// TIA Portal project "EdgeHowTos_V19" (V19)

(* hardware
DEVICE "S71500/ET200MP station_1"  S7-1500 station
   slot 0: "Rail_0"  Rack  6ES7 590-1***0-0AA0
   slot 1: "Tank application"  CPU 1513-1 PN  6ES7 513-1AL02-0AB0  V2.8
      slot 3: "CPU display_1"  6ES7591-1AA00-0AA0
      slot 32768: "PROFINET interface_1"  X1
         slot 32769: "Port_1"  X1 P1
         slot 32770: "Port_2"  X1 P2
      slot 34817: "Virtual CP interface port_1"  Virtual CP interface port  Virtual CP interface port
DEVICE "TP900"  TP900 Comfort
   slot 0: "TP900"  TP900 Comfort  6AV2 124-0JC01-0AX0  16.0.0.0
   slot 1: "HMI_RT_5"  TP900 Comfort  6AV2 124-0JC01-0AX0  16.0.0.0
   slot 5: "TP900._CP_1"  PROFINET Interface  16.0.0.0
      slot 1: "PROFINET Interface_1"  PROFINET Interface
         slot 1: "Port_1"  Port
         slot 2: "Port_2"  Port
   slot 7: "TP900.I/DP_CP_1"  MPI/DP Interface  16.0.0.0
DEVICE "MTP1500"  MTP1500 Unified Comfort
   slot 0: "0"  MTP1500 Unified Comfort  6AV2 128-3QB06-0AXx  19.0.0.0
   slot 1: "MTP1500_Runtime"  MTP1500 Unified Comfort  6AV2 128-3QB06-0AXx  19.0.0.0
   slot 5: "0.IE_CP_1"  PROFINET Interface  19.0.0.0
      slot 1: "PROFINET Interface_1"  PROFINET Interface
         slot 1: "Port_1"  Port
         slot 2: "Port_2"  Port
   slot 6: "0.IE_CP_2"  PROFINET Interface  19.0.0.0
      slot 1: "PROFINET Interface_GBit"  PROFINET Interface
         slot 1: "Port_1"  Port
*)

// ===== PLC "Tank application"  CPU 1513-1 PN =====

VAR_GLOBAL   // PLC tag table "Default tag table"
   "Manipulator" AT %MW0 : Int;
END_VAR

VAR_GLOBAL CONSTANT   // PLC tag table "Default tag table"
   "STATE_FILL_TANK" : Int := 1;
   "STATE_HEAT_TANK" : Int := 2;
   "STATE_FILL_BOTTLE" : Int := 3;
   "STATE_SHIFT_BOTTLE" : Int := 4;
   "STATE_STOP" : Int := 5;
   "STATE_RESET" : Int := 6;
   "STATE_ERROR" : Int := 7;
   "ERROR_0_NoError" : UInt := 8000;
   "ERROR_1_BottleInWrongPosition" : UInt := 8001;
   "ERROR_2_CrackedBottleDetected" : UInt := 8002;
   "ERROR_3_NoBottleOnTheConveyor" : UInt := 8003;
   "ERROR_4_WrongBottleDetected" : UInt := 8004;
   "ERROR_5_ConveyorMalfunction" : UInt := 8005;
   "ERROR_6_FillerMalfunction" : UInt := 8006;
   "ERROR_7_ValveBlocked" : UInt := 8007;
   "ERROR_8_NoFlowInMainPipe" : UInt := 8008;
   "ERROR_9_GenericError_CheckPlcBuffer" : UInt := 8009;
   "ERROR_10_GenericError_CheckAlarmBuffer" : UInt := 8010;
   "ERROR_11_GenericError_ContactWithSupplier" : UInt := 8011;
   "OEE_ERROR_1_BottleInWrongPosition" : UInt := 4;
   "OEE_ERROR_10_GenericError_CheckAlarmBuffer" : UInt := 13;
   "OEE_ERROR_11_GenericError_ContactWithSupplier" : UInt := 14;
   "OEE_ERROR_2_CrackedBottleDetected" : UInt := 5;
   "OEE_ERROR_3_NoBottleOnTheConveyor" : UInt := 6;
   "OEE_ERROR_4_WrongBottleDetected" : UInt := 7;
   "OEE_ERROR_5_ConveyorMalfunction" : UInt := 8;
   "OEE_ERROR_6_FillerMalfunction" : UInt := 9;
   "OEE_ERROR_7_ValveBlocked" : UInt := 10;
   "OEE_ERROR_8_NoFlowInMainPipe" : UInt := 11;
   "OEE_ERROR_9_GenericError_CheckPlcBuffer" : UInt := 12;
   "OEE_PRODUCTION" : UInt := 1;
   "OEE_PLANNED_DOWN" : UInt := 2;
   "OEE_UNPLANNED_DOWN" : UInt := 3;
END_VAR

TYPE "typeHmi"
   STRUCT
      HMI_Start : Bool;   // trigger from hmi to start
      HMI_Stop : Bool;   // trigger from hmi to stop
      HMI_Reset : Bool;   // trigger from hmi to reset
      HMI_NextBottle : Bool;   // trigger from hmi to shift bottle
      HMI_Error : Bool;   // trigger from hmi to generate error
      HMI_InstallFillingPump : Bool;   // trigger from hmi to install filling pump
      HMI_RenewHeatingElement : Bool;   // trigger from hmi to renew heating element
   END_STRUCT;
END_TYPE

TYPE "typeApp"
   STRUCT
      APP_Start : Bool;   // trigger from app to start
      APP_Stop : Bool;   // trigger from app to stop
      APP_Reset : Bool;   // trigger from app to reset
      APP_QRCode : String;   // string from app containing QR code (scanning app)
      APP_ErrorSimulation : Bool;   // activate automatically error simulation (true = active)
      APP_Error : Bool;   // generate a manual error (true = error)
      APP_Alarm : Bool;   // trigger from app to generate program alarm
   END_STRUCT;
END_TYPE

TYPE "typeSignals"
   STRUCT
      tankSignals : Struct
         actLevel : Real;   // actual level of tank [l]
         maxLevel : Bool;   // max level of tank reached
         actPressure : Real;   // actual pressure of tank [hPa]
         actTemperature : Real;   // actual temperature of tank [°C]
         maxTemperature : Bool;   // max level of temperature reached
      END_STRUCT;
      bottleSignals : Struct
         actLevel : Real;   // actual level of current bottle [l]
         maxLevel : Bool;   // max level of bottle reached
         outputTank : Real;   // Vout of Tank / Vin of bottle [m³/s]
      END_STRUCT;
      energySignals : Struct
         energyConsumptionFillingTank : Real;   // energy consumption during filling tank [Wh]
         waterConsumptionFillingTank : Real;   // water consumption during filling tank [l]
         energyConsumptionHeatingTank : Real;   // energy consumption during heating tank [Wh]
         energyConsumptionFillingBottles : Real;   // energy consumption during filling bottles [Wh]
         gasConsumptionHeatingTank : Real;   // gas consumption during heating tank [Wh]
      END_STRUCT;
      energySignalsPerState : Struct
         stateId : UInt;   // ID per standart state
         energyConsumptionStatePoweringUp : Real;   // energy consumption during state powering up [kWh]
         energyConsumptionStatePoweringDown : Real;   // energy consumption during state powering down [kWh]
         energyConsumptionStateOff : Real;   // energy consumption during state off [kWh]
         energyConsumptionStateStandby : Real;   // energy consumption during state standby [kWh]
         energyConsumptionStateOperational : Real;   // energy consumption during state operational [kWh]
         energyConsumptionStateWorking : Real;   // energy consumption during state working [kWh]
         energyConsumptionStatesTotal : Real;   // total energy consumption of states [kWh]
      END_STRUCT;
      alarm : Word;   // alarm bit
      errorCode : UInt;   // error code
   END_STRUCT;
END_TYPE

TYPE "typeOperate"
   STRUCT
      extModeActive : Bool := false;   // true = activate external model / simulation
      state : "typeState";   // operating state
      machineState : Int := 0;   // machine production state (1 = filling tank, 2 = heating tank, 3 = filling bottle, 4 = shifting bottle, 5 = stop, 6 = reset)
      machineStateOEE : Int := 0;   // machine OEE state (1 = production, 2 = planned downtime, 3 = unplanned downtime)
   END_STRUCT;
END_TYPE

TYPE "typeModel"
   STRUCT
      cycleTime : Real;   // cycle time[s]
      tank : Struct   // model struct of tank
         AT : Real;   // surface area of tank [m²]
         H : Real;   // high of tank [m]
         Vin : Real;   // incoming volume flow [l/min]
         maxLevel : Real;   // max level of tank [m³]
         roomTemperature : Real;   // room temperature of tank [°C]
         maxTemperature : Real;   // max temperature of tank [°C]
         density : Real;   // liquid density [kg/m³]
      END_STRUCT;
      bottle : Struct   // model struct of bottle
         maxLevel : Real;   // max level of bottle [m³]
         AB : Real;   // surface area of filling hole to fill bottle [m²]
         shiftingCycle : UInt;   // bottle shifting cycle
      END_STRUCT;
   END_STRUCT;
END_TYPE

TYPE "typeProcess"
   STRUCT
      productId : String;   // product id of current bottle
      numberProduced : UDInt;   // number of filled bottles
      numberFaulty : UDInt;   // number of faulty bottles
      numberGood : UDInt;   // number of good bottles
      batchId : UDInt;   // batch id (according to tank filling)
      productTypeId : UInt;   // type id - for generating of the serial number and QR code
      productTypeName : String;   // type name of product
      productSerialNumber : String;   // serial number per product
      productQRCode : USInt;   // qr code per product
      speedActual : UDInt;   // actual production speed (pcs/h)
      speedTarget : UDInt;   // target production speed (pcs/h)
   END_STRUCT;
END_TYPE

TYPE "typeState"
   STRUCT
      FillingTank : Bool;   // filling tank
      HeatingTank : Bool;   // heating tank
      FillingBottle : Bool;   // filling bottle
      ShiftingBottle : Bool;   // shifting bottle
      Stop : Bool;   // stop filling application
      Reset : Bool;   // reset application
      Error : Bool;   // error within filling application
   END_STRUCT;
END_TYPE

TYPE "typeInfo"
   STRUCT
      "version" : String;   // current version of the project
      "date" : String;   // last change date of the project
   END_STRUCT;
END_TYPE

TYPE "typeError"
   STRUCT
      errorTrigger : Bool := false;   // manually trigger error simulation
      errorDuration : Time := T#300s;   // error duration for simulation
   END_STRUCT;
END_TYPE

TYPE "typeCIP"
   STRUCT
      cipStartTime : Time_Of_Day := TOD#22:00:00;   // CIP start time 1x per day
      cipActive : Bool;   // Activate/deactivate the CIP process
      cipId : Int;   // CIP id
      cipProcess : String;   // CIP process (full wash, quick wash)
      cipStep : String;   // CIP step
      cipTemperature : Real;   // CIP temperature
      cipConcentration : Real;   // CIP concentration
      cipFlowrate : Real;   // CIP flowrate
      cipStep1 : Bool;   // Step 1 active
      cipStep2 : Bool;   // Step 2 active
      cipStep3 : Bool;   // Step 3 active
      cipStep4 : Bool;   // Step 4 active
   END_STRUCT;
END_TYPE

DATA_BLOCK "GDB"   // DB1
{ S7_Optimized_Access := 'FALSE' }
VERSION : 0.1
   VAR
      operate : "typeOperate";   // application operation
      model : "typeModel";   // model parameter
      externalSignals : "typeSignals";   // signals from external model
      signals : "typeSignals";   // current signals from tank and bottle
      process : "typeProcess";   // current process information
      hmiSignals : "typeHmi";   // signals from hmi
      appSignals : "typeApp";   // signals from edge app
      projectInfo : "typeInfo";   // infos regarding this TIA project
      errors : "typeError";   // parameter for error simulation
      cip : "typeCIP";   // parameter for cip simulation (tank cleaning)
   END_VAR
BEGIN
   model.tank.H := 2.0;
   model.tank.AT := 0.8;
   operate.extModeActive := false;
   model.tank.maxTemperature := 80.0;
   model.tank.maxLevel := 1.6;
   model.bottle.maxLevel := 0.001;
   model.cycleTime := 0.005;
   model.tank.roomTemperature := 20.0;
   model.tank.Vin := 500.0;
   model.bottle.AB := 5.0E-06;
   process.productId := '';
   process.numberProduced := 0;
   process.numberFaulty := 0;
   model.tank.density := 997.0;
   hmiSignals.HMI_Start := true;
   projectInfo."version" := 'V4.0';
   projectInfo."date" := '2025-07-01';
   errors.errorDuration := T#10m;
   model.bottle.shiftingCycle := 50;
   appSignals.APP_ErrorSimulation := true;
   process.speedActual := 3700;
   process.speedTarget := 4000;
END_DATA_BLOCK

DATA_BLOCK "DB_1_Sequence"   // DB2
{ S7_Optimized_Access := 'TRUE' }
VERSION : 0.1
// stored: InstanceOfName FB_1_Sequence
"FB_1_Sequence"
BEGIN
END_DATA_BLOCK

DATA_BLOCK "DB_2_Filling_DB"   // DB3
{ S7_Optimized_Access := 'TRUE' }
VERSION : 0.1
// stored: InstanceOfName FB_2_Filling
"FB_2_Filling"
BEGIN
END_DATA_BLOCK

DATA_BLOCK "DB_3_Simulation"   // DB4
{ S7_Optimized_Access := 'TRUE' }
VERSION : 0.1
// stored: InstanceOfName FB_3_Simulation
"FB_3_Simulation"
BEGIN
END_DATA_BLOCK

DATA_BLOCK "Generate_Serial_Number_DB"   // DB6
{ S7_Optimized_Access := 'TRUE' }
VERSION : 0.1
// stored: InstanceOfName FB_Generate_Serial_Number
"FB_Generate_Serial_Number"
BEGIN
END_DATA_BLOCK

DATA_BLOCK "Block_1_DB"   // DB7
{ S7_Optimized_Access := 'TRUE' }
VERSION : 0.1
// stored: InstanceOfName FB_Prodiag
"FB_Prodiag"
BEGIN
END_DATA_BLOCK

DATA_BLOCK "DB_4_CIP_Simulation"   // DB11
{ S7_Optimized_Access := 'TRUE' }
VERSION : 0.1
// stored: InstanceOfName FB_4_CIP_Simulation
"FB_4_CIP_Simulation"
BEGIN
END_DATA_BLOCK

DATA_BLOCK "DB_5_CIP_Simulation_Graph"   // DB14
{ S7_Optimized_Access := 'TRUE' }
VERSION : 0.1
// stored: InstanceOfName FB_5_CIP_Simulation_Graph
"FB_5_CIP_Simulation_Graph"
BEGIN
END_DATA_BLOCK

// folder: System blocks/Program resources

DATA_BLOCK "IEC_Timer_CIP_Step2"   // DB12
{ S7_Optimized_Access := 'TRUE' }
AUTHOR : Simatic
FAMILY : IEC
NAME : IEC_TMR
VERSION : 1.0
// stored: InstanceOfName IEC_TIMER
"IEC_TIMER"
BEGIN
END_DATA_BLOCK

DATA_BLOCK "IEC_Timer_CIP_Init"   // DB15
{ S7_Optimized_Access := 'TRUE' }
AUTHOR : Simatic
FAMILY : IEC
NAME : IEC_TMR
VERSION : 1.0
// stored: InstanceOfName IEC_TIMER
"IEC_TIMER"
BEGIN
END_DATA_BLOCK

DATA_BLOCK "IEC_Timer_CIP_Step3"   // DB20
{ S7_Optimized_Access := 'TRUE' }
AUTHOR : Simatic
FAMILY : IEC
NAME : IEC_TMR
VERSION : 1.0
// stored: InstanceOfName IEC_TIMER
"IEC_TIMER"
BEGIN
END_DATA_BLOCK

DATA_BLOCK "IEC_Timer_CIP_Step4"   // DB21
{ S7_Optimized_Access := 'TRUE' }
AUTHOR : Simatic
FAMILY : IEC
NAME : IEC_TMR
VERSION : 1.0
// stored: InstanceOfName IEC_TIMER
"IEC_TIMER"
BEGIN
END_DATA_BLOCK

DATA_BLOCK "IEC_Timer_CIP_End"   // DB22
{ S7_Optimized_Access := 'TRUE' }
AUTHOR : Simatic
FAMILY : IEC
NAME : IEC_TMR
VERSION : 1.0
// stored: InstanceOfName IEC_TIMER
"IEC_TIMER"
BEGIN
END_DATA_BLOCK

// folder: (top level)

FUNCTION_BLOCK "FB_Generate_Serial_Number"   // FB1, LAD
{ S7_Optimized_Access := 'TRUE' }
VERSION : 0.1
   VAR_INPUT
      batchId : UDInt;
      productId : UDInt;
      productType : Int;
      trigger : Bool;
   END_VAR
   VAR_OUTPUT
      serialNumber : String;
      qrCode : USInt;
   END_VAR
   VAR
      sizeBatch : USInt;
      sizeId : USInt;
      retVal : USInt;
      dateString : String;
      batchString : String;
      productString : String;
      typeString : String;
      pTrigAux_1 : Bool;
   END_VAR
   VAR_TEMP
      localTime : DTL;
      qrNoTemp : String;
   END_VAR
   VAR_TEMP   // added for the SCL form of the ladder/FBD networks
      _w1 : Bool;
   END_VAR
BEGIN

REGION Network 1 (SCL)
   // get string size of batch ID
   "FC_2_GetStringSizeOfNumber"(number:=#batchId,
                                stringSize=>#sizeBatch);

   // get string size of prodcut ID
   "FC_2_GetStringSizeOfNumber"(number:=#productId,
                                stringSize=>#sizeId);
END_REGION

REGION Network 2
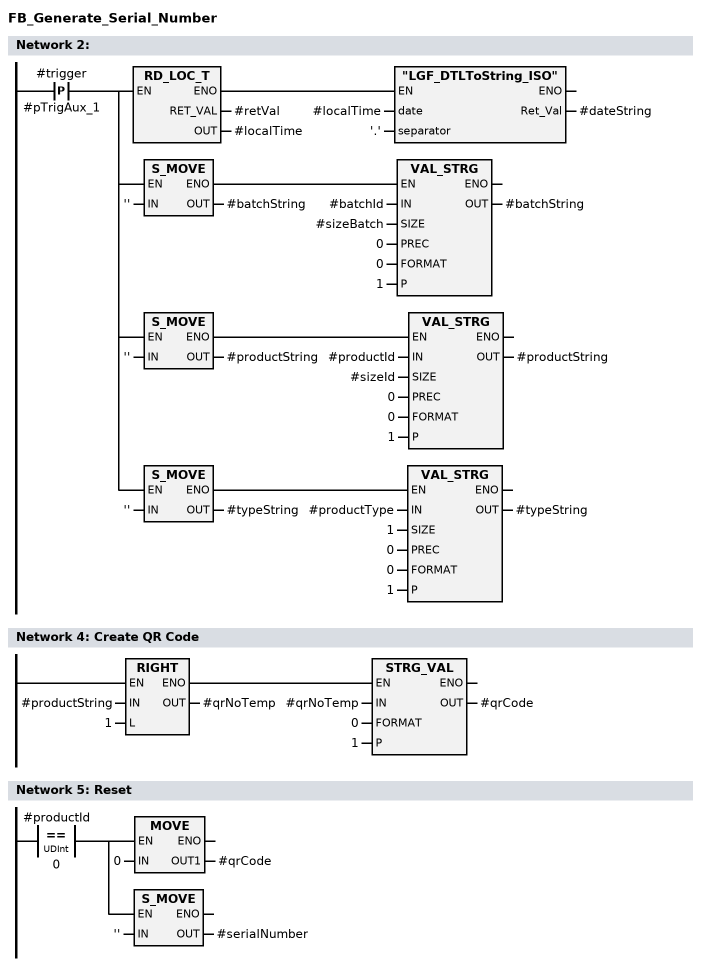
   // ENO of a box is taken as its EN; it also drops when the box reports an error
   #_w1 := #trigger AND NOT #pTrigAux_1;   // rising edge of #trigger
   #pTrigAux_1 := #trigger;
   IF #_w1 THEN
       #retVal := RD_LOC_T(OUT => #localTime);
       #dateString := "LGF_DTLToString_ISO"("date" := #localTime, separator := '.');
       #batchString := '';
       VAL_STRG(IN := #batchId, SIZE := #sizeBatch, PREC := 0, FORMAT := 0, P := 1, OUT => #batchString);
       #productString := '';
       VAL_STRG(IN := #productId, SIZE := #sizeId, PREC := 0, FORMAT := 0, P := 1, OUT => #productString);
       #typeString := '';
       VAL_STRG(IN := #productType, SIZE := 1, PREC := 0, FORMAT := 0, P := 1, OUT => #typeString);
   END_IF;
END_REGION

REGION Network 3 (SCL): Create serial number
   #serialNumber := CONCAT(
                            IN1 := REPLACE(IN1:=DELETE(IN:=#dateString, L:=13, P:=17), IN2:='/', L:=1, P:=11),
                            IN2 := '/',
                            IN3 := #typeString,
                            IN4 := '/',
                            IN5 := #batchString,
                            IN6 := '/',
                            IN7 := #productString
   );
END_REGION

REGION Network 4: Create QR Code
   #qrNoTemp := RIGHT(IN := #productString, L := 1);
   STRG_VAL(IN := #qrNoTemp, FORMAT := 0, P := 1, OUT => #qrCode);
END_REGION

REGION Network 5: Reset
   RUNG wire#powerrail
      { S7_Templates := "SrcType := UDInt" } EQ_Contact(in1 := #productId, in2 := 0)
      wire#w1
      Move(in := 0, out1 => #qrCode)
   END_RUNG
   RUNG wire#w1
      S_Move(in := '', out => #serialNumber)
   END_RUNG
   // the same network as SCL:
   IF #productId = 0 THEN
       #qrCode := 0;
       #serialNumber := '';
   END_IF;
END_REGION
END_FUNCTION_BLOCK

FUNCTION_BLOCK "FB_1_Sequence"   // FB2, FBD
{ S7_Optimized_Access := 'TRUE' }
VERSION : 0.1
   VAR_INPUT
      externalSignals : "typeSignals";   // signals from external model
   END_VAR
   VAR_IN_OUT
      model : "typeModel";   // model parameter
      operate : "typeOperate";   // application operation
      signals : "typeSignals";   // current signals from tank
      process : "typeProcess";   // current process information
      hmi : "typeHmi";   // signals from hmi
      app : "typeApp";   // signals from app
      errors : "typeError";
   END_VAR
   VAR
      statStart : Bool;   // trigger for start command
      statStop : Bool;   // trigger for stop command
      statReset : Bool;   // trigger for reset command
      statInit : Bool := true;   // helper variable to initialize some parameters
      statNextBottle : Bool;   // trigger to shift next bottle
      statError : Bool;   // trigger to set error
      statState : Int;   // memory for reactivating state after STOP
      statAlarm : Bool;   // trigger to generate program alarm
      statMemoryStart : Bool;
      statMemoryStop : Bool;
      statMemoryReset : Bool;
      statMemoryNextBottle : Bool;
      statMemoryError : Bool;
      statHmiStateStart : Bool;   // helper for hmi (true, if state 1-4)
      statShiftingTimer : Int;
      statShiftingTimerTrigger : Bool;
      statShiftingTrigger : Bool;
      statShiftingTimerDone : Bool;
      statHmiQrCodeReceived : Bool;
      statHMIQrCodeReceivedTrigger : Bool;
      statQrCodeTrigger : Bool;
      statTankEmpty : Bool;   // trigger when tank is empty
      statTankEmptyMemory : Bool;   // tank empty memory
      statOverflow : Bool;   // overflow of counter "numberProduced"
      statOverflowStartTrigger : Bool;   // trigger to start after overflow
      statOverflowStartMemory : Bool;
      Program_Alarm : Program_Alarm;
      statAssocValues : AssocValues;   // values for Gen_UsrMsg block
      statTriggerAlarm : Bool;
      statTriggerAlarmMemory : Bool;
      statErrorCodeOld : UInt;
   END_VAR
   VAR_TEMP
      tempQrCodeLen : Int;
      tempProgramAlarmError : Bool;
      tempProgramAlarmStatus : Word;
      tempAlarmStateError : Bool;
      tempAlarmStateStatus : Word;
      tempProgramAlarmError2 : Bool;
      tempProgramAlarmStatus2 : Word;
      tempAlarmStateError2 : Bool;
      tempAlarmStateStatus2 : Word;
      tempRetVal : Int;
   END_VAR
   VAR_TEMP   // added for the SCL form of the ladder/FBD networks
      _w1 : Bool;
      _w2 : Bool;
      _w3 : Bool;
   END_VAR
BEGIN

REGION Network 1: Handling signals from hmi or app
   // --[P]-- (positive signal edge) -> stat-Variable becomes true for one cycle
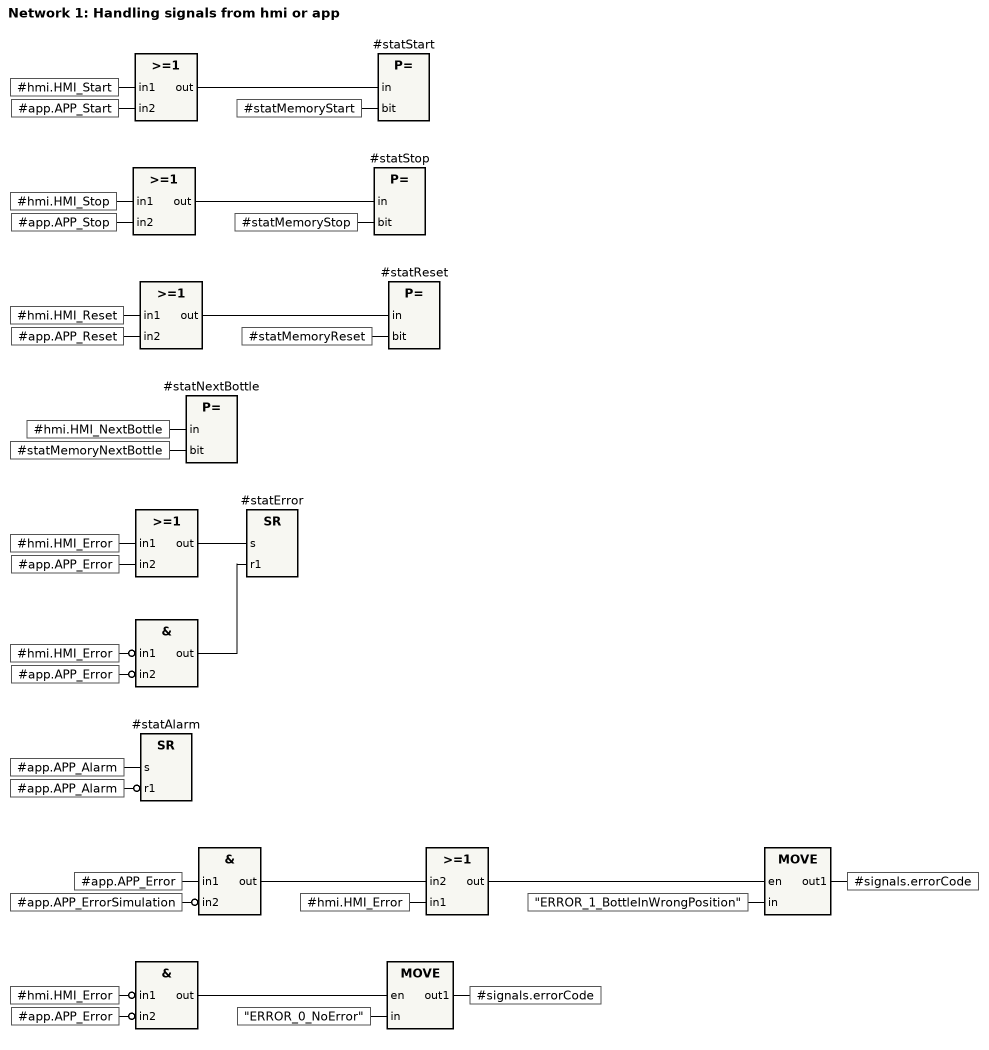
   #_w1 := #hmi.HMI_Start OR #app.APP_Start;
   #statStart := #_w1 AND NOT #statMemoryStart;   // rising edge
   #statMemoryStart := #_w1;
   #_w2 := #hmi.HMI_Stop OR #app.APP_Stop;
   #statStop := #_w2 AND NOT #statMemoryStop;   // rising edge
   #statMemoryStop := #_w2;
   #_w3 := #hmi.HMI_Reset OR #app.APP_Reset;
   #statReset := #_w3 AND NOT #statMemoryReset;   // rising edge
   #statMemoryReset := #_w3;
   #statNextBottle := #hmi.HMI_NextBottle AND NOT #statMemoryNextBottle;   // rising edge
   #statMemoryNextBottle := #hmi.HMI_NextBottle;
   IF #hmi.HMI_Error OR #app.APP_Error THEN
       #statError := TRUE;   // SR flip-flop
   END_IF;
   IF NOT #hmi.HMI_Error AND NOT #app.APP_Error THEN #statError := FALSE; END_IF;
   IF #app.APP_Alarm THEN
       #statAlarm := TRUE;   // SR flip-flop
   END_IF;
   IF NOT #app.APP_Alarm THEN #statAlarm := FALSE; END_IF;
   IF (#app.APP_Error AND NOT #app.APP_ErrorSimulation) OR #hmi.HMI_Error THEN
       #signals.errorCode := "ERROR_1_BottleInWrongPosition";
   END_IF;
   IF NOT #hmi.HMI_Error AND NOT #app.APP_Error THEN #signals.errorCode := "ERROR_0_NoError"; END_IF;
END_REGION

REGION Network 2: Reset signals from hmi or app
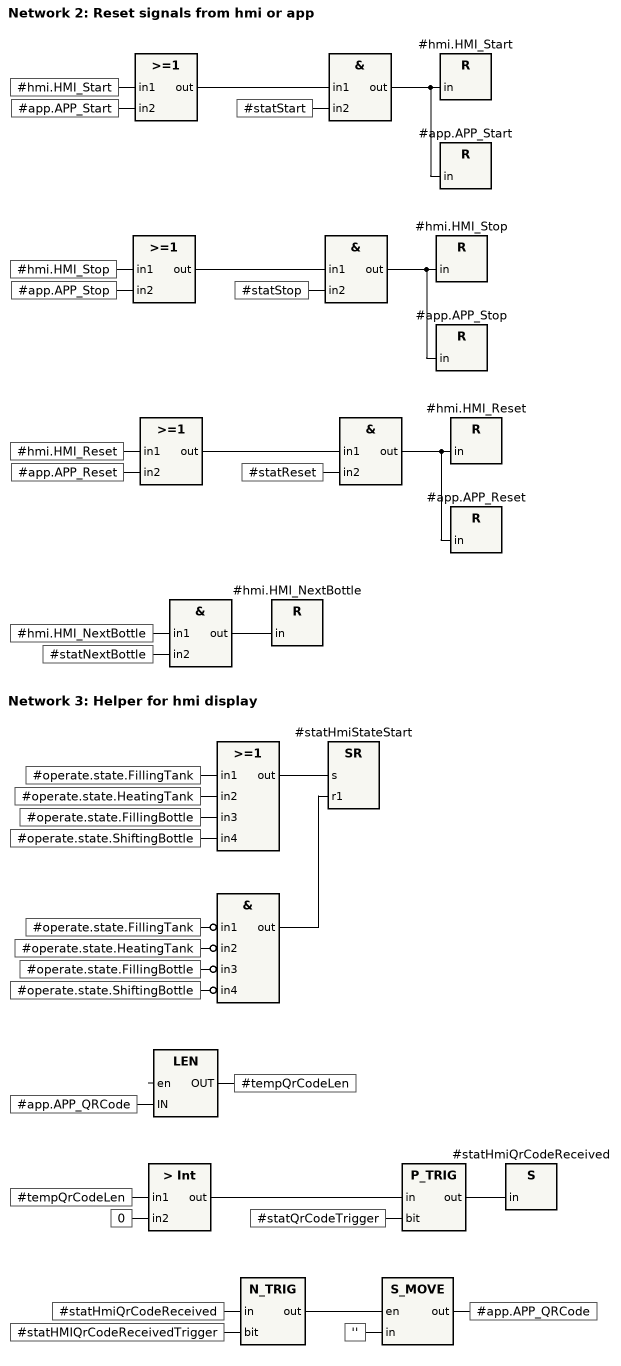
   #_w1 := (#hmi.HMI_Start OR #app.APP_Start) AND #statStart;
   IF #_w1 THEN
       #hmi.HMI_Start := FALSE;
       #app.APP_Start := FALSE;
   END_IF;
   #_w2 := (#hmi.HMI_Stop OR #app.APP_Stop) AND #statStop;
   IF #_w2 THEN
       #hmi.HMI_Stop := FALSE;
       #app.APP_Stop := FALSE;
   END_IF;
   #_w3 := (#hmi.HMI_Reset OR #app.APP_Reset) AND #statReset;
   IF #_w3 THEN
       #hmi.HMI_Reset := FALSE;
       #app.APP_Reset := FALSE;
   END_IF;
   IF #hmi.HMI_NextBottle AND #statNextBottle THEN #hmi.HMI_NextBottle := FALSE; END_IF;
END_REGION

REGION Network 3: Helper for hmi display
   IF #operate.state.FillingTank OR #operate.state.HeatingTank OR #operate.state.FillingBottle OR #operate.state.ShiftingBottle THEN
       #statHmiStateStart := TRUE;   // SR flip-flop
   END_IF;
   IF NOT #operate.state.FillingTank AND NOT #operate.state.HeatingTank AND NOT #operate.state.FillingBottle AND NOT #operate.state.ShiftingBottle THEN
       #statHmiStateStart := FALSE;
   END_IF;
   #tempQrCodeLen := LEN(IN := #app.APP_QRCode);
   #_w1 := #tempQrCodeLen > 0;
   #_w2 := #_w1 AND NOT #statQrCodeTrigger;   // rising edge
   #statQrCodeTrigger := #_w1;
   IF #_w2 THEN #statHmiQrCodeReceived := TRUE; END_IF;
   #_w3 := NOT #statHmiQrCodeReceived AND #statHMIQrCodeReceivedTrigger;   // falling edge
   #statHMIQrCodeReceivedTrigger := #statHmiQrCodeReceived;
   IF #_w3 THEN #app.APP_QRCode := ''; END_IF;
END_REGION

REGION Network 4: SHIFTING: shifting bottle - timer
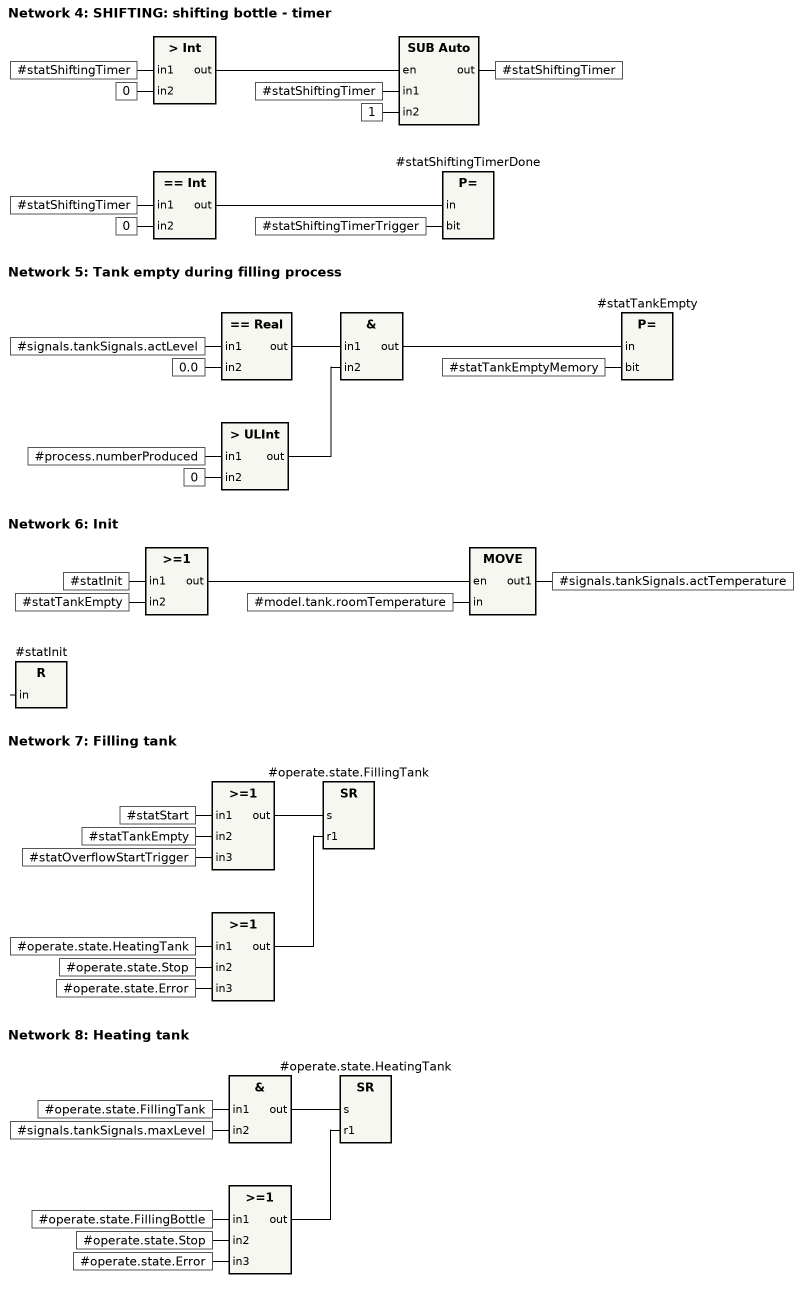
   IF #statShiftingTimer > 0 THEN #statShiftingTimer := #statShiftingTimer - 1; END_IF;
   #_w1 := #statShiftingTimer = 0;
   #statShiftingTimerDone := #_w1 AND NOT #statShiftingTimerTrigger;   // rising edge
   #statShiftingTimerTrigger := #_w1;
END_REGION

REGION Network 5: Tank empty during filling process
   #_w1 := (#signals.tankSignals.actLevel = 0.0) AND (#process.numberProduced > 0);
   #statTankEmpty := #_w1 AND NOT #statTankEmptyMemory;   // rising edge
   #statTankEmptyMemory := #_w1;
END_REGION

REGION Network 6: Init
   IF #statInit OR #statTankEmpty THEN
       #signals.tankSignals.actTemperature := #model.tank.roomTemperature;
   END_IF;
   #statInit := FALSE;
END_REGION

REGION Network 7: Filling tank
   IF #statStart OR #statTankEmpty OR #statOverflowStartTrigger THEN
       #operate.state.FillingTank := TRUE;   // SR flip-flop
   END_IF;
   IF #operate.state.HeatingTank OR #operate.state.Stop OR #operate.state.Error THEN
       #operate.state.FillingTank := FALSE;
   END_IF;
END_REGION

REGION Network 8: Heating tank
   IF #operate.state.FillingTank AND #signals.tankSignals.maxLevel THEN
       #operate.state.HeatingTank := TRUE;   // SR flip-flop
   END_IF;
   IF #operate.state.FillingBottle OR #operate.state.Stop OR #operate.state.Error THEN
       #operate.state.HeatingTank := FALSE;
   END_IF;
END_REGION

REGION Network 9: Filling bottle
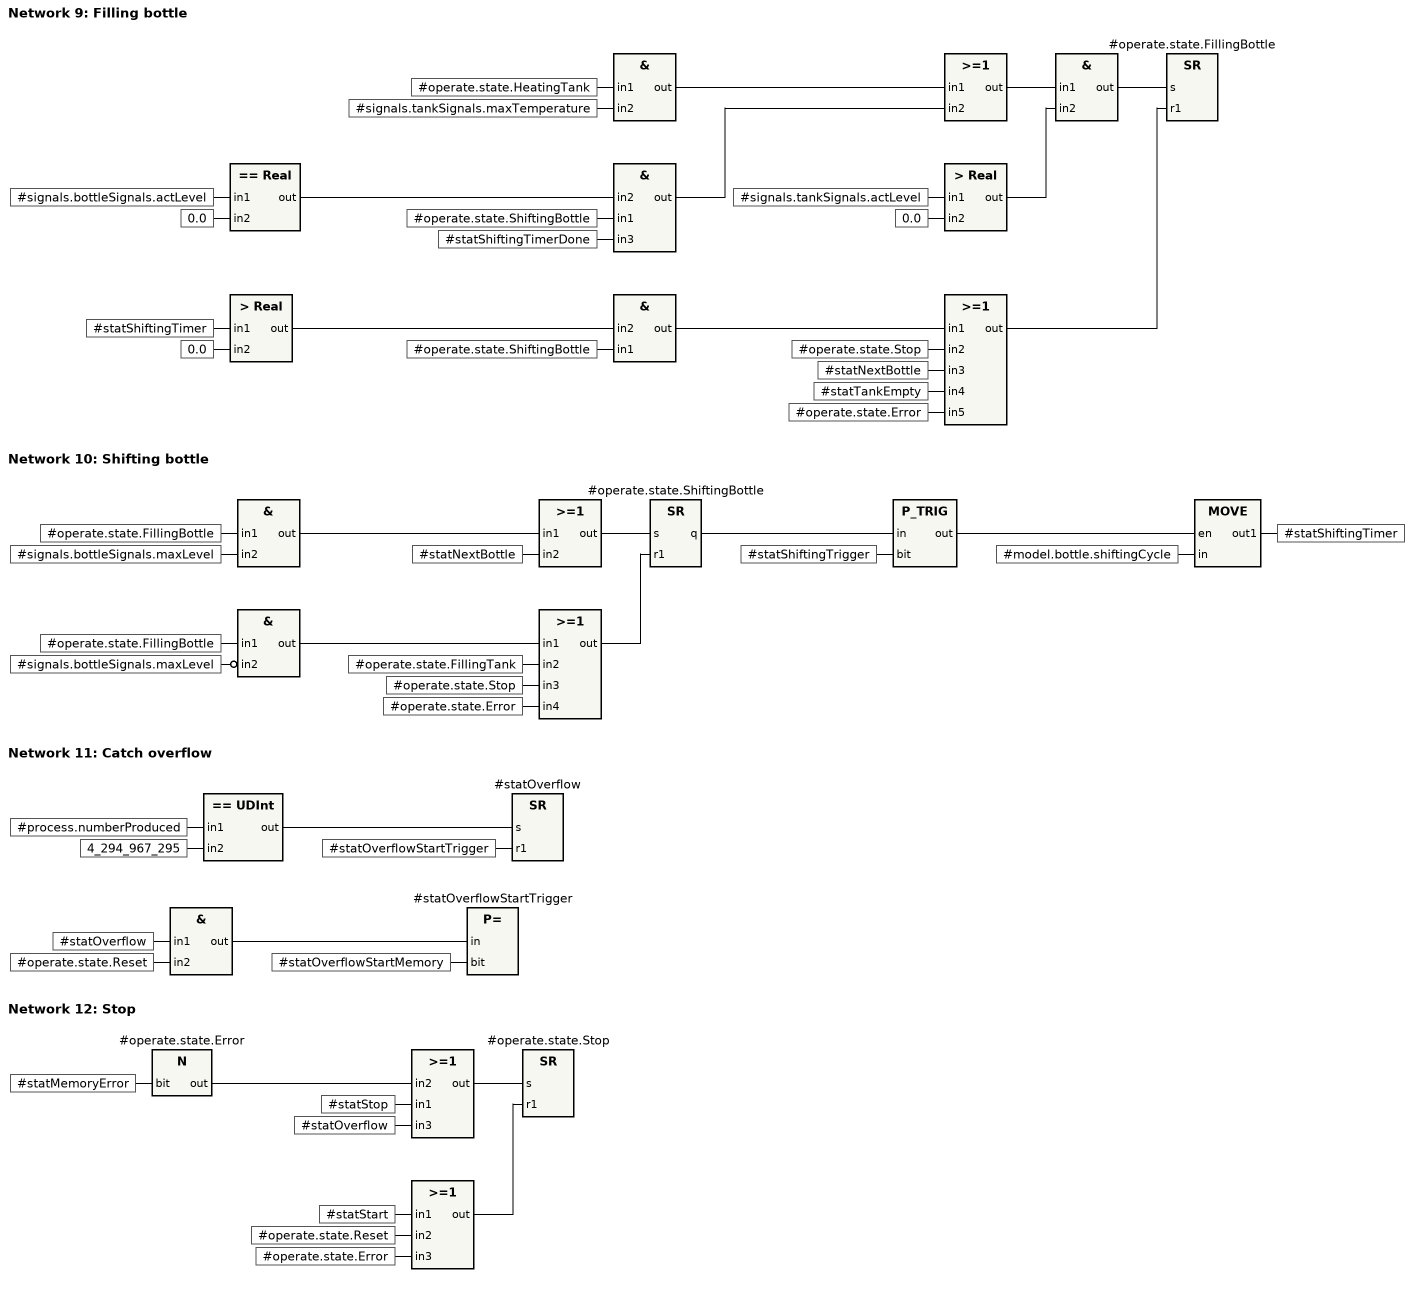
   IF ((#operate.state.HeatingTank AND #signals.tankSignals.maxTemperature) OR ((#signals.bottleSignals.actLevel = 0.0) AND #operate.state.ShiftingBottle AND #statShiftingTimerDone)) AND (#signals.tankSignals.actLevel > 0.0) THEN
       #operate.state.FillingBottle := TRUE;   // SR flip-flop
   END_IF;
   IF ((#statShiftingTimer > 0.0) AND #operate.state.ShiftingBottle) OR #operate.state.Stop OR #statNextBottle OR #statTankEmpty OR #operate.state.Error THEN
       #operate.state.FillingBottle := FALSE;
   END_IF;
END_REGION

REGION Network 10: Shifting bottle
   IF (#operate.state.FillingBottle AND #signals.bottleSignals.maxLevel) OR #statNextBottle THEN
       #operate.state.ShiftingBottle := TRUE;   // SR flip-flop
   END_IF;
   IF (#operate.state.FillingBottle AND NOT #signals.bottleSignals.maxLevel) OR #operate.state.FillingTank OR #operate.state.Stop OR #operate.state.Error THEN
       #operate.state.ShiftingBottle := FALSE;
   END_IF;
   #_w1 := #operate.state.ShiftingBottle AND NOT #statShiftingTrigger;   // rising edge
   #statShiftingTrigger := #operate.state.ShiftingBottle;
   IF #_w1 THEN #statShiftingTimer := #model.bottle.shiftingCycle; END_IF;
END_REGION

REGION Network 11: Catch overflow
   // If max of UDINT is reached
   // > Stop (automatically)
   // > Reset (automatically)
   // > Start (automatically)
   IF #process.numberProduced = 4_294_967_295 THEN
       #statOverflow := TRUE;   // SR flip-flop
   END_IF;
   IF #statOverflowStartTrigger THEN #statOverflow := FALSE; END_IF;
   #_w1 := #statOverflow AND #operate.state.Reset;
   #statOverflowStartTrigger := #_w1 AND NOT #statOverflowStartMemory;   // rising edge
   #statOverflowStartMemory := #_w1;
END_REGION

REGION Network 12: Stop
   #_w1 := NOT #operate.state.Error AND #statMemoryError;   // falling edge of #operate.state.Error
   #statMemoryError := #operate.state.Error;
   IF #_w1 OR #statStop OR #statOverflow THEN
       #operate.state.Stop := TRUE;   // SR flip-flop
   END_IF;
   IF #statStart OR #operate.state.Reset OR #operate.state.Error THEN #operate.state.Stop := FALSE; END_IF;
END_REGION

REGION Network 13: Reset
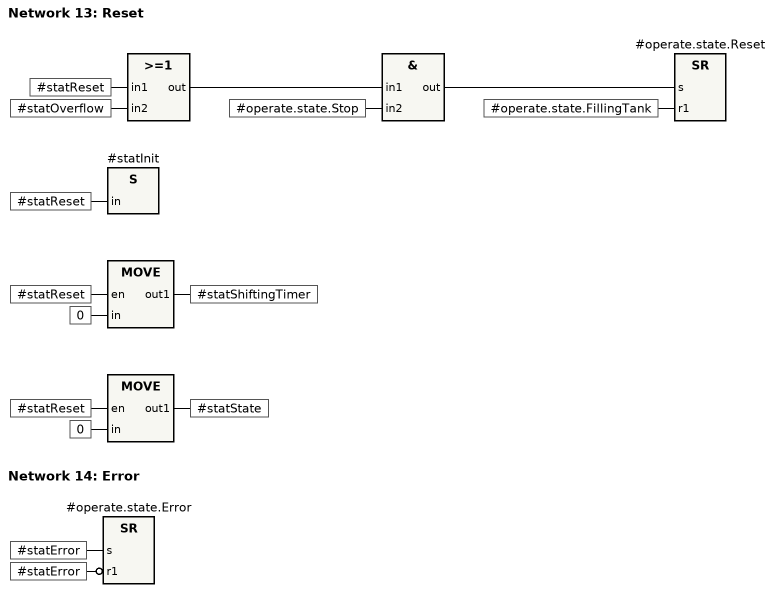
   IF (#statReset OR #statOverflow) AND #operate.state.Stop THEN
       #operate.state.Reset := TRUE;   // SR flip-flop
   END_IF;
   IF #operate.state.FillingTank THEN #operate.state.Reset := FALSE; END_IF;
   IF #statReset THEN
       #statInit := TRUE;
       #statShiftingTimer := 0;
       #statState := 0;
   END_IF;
END_REGION

REGION Network 14: Error
   IF #statError THEN
       #operate.state.Error := TRUE;   // SR flip-flop
   END_IF;
   IF NOT #statError THEN #operate.state.Error := FALSE; END_IF;
END_REGION

REGION Network 15: Set machine state
   // 1 = filling tank
   // 2 = heating tank
   // 3 = filling bottle
   // 4 = shifting bottle
   // 5 = stop
   // 6 = reset
   // 7 = error
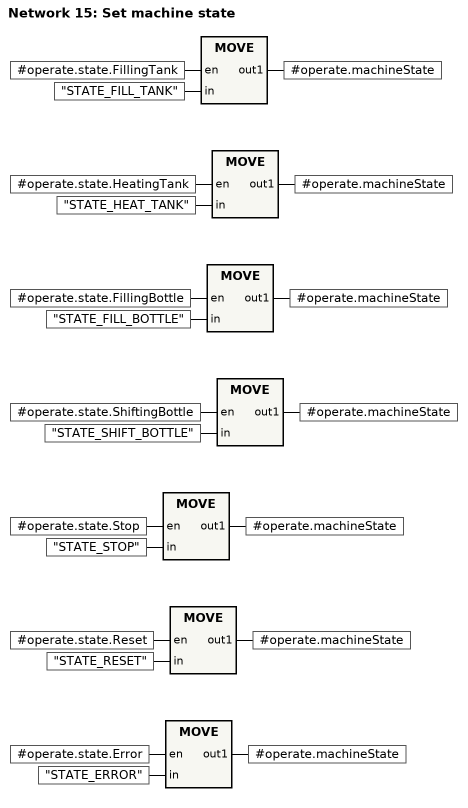
   IF #operate.state.FillingTank THEN #operate.machineState := "STATE_FILL_TANK"; END_IF;
   IF #operate.state.HeatingTank THEN #operate.machineState := "STATE_HEAT_TANK"; END_IF;
   IF #operate.state.FillingBottle THEN #operate.machineState := "STATE_FILL_BOTTLE"; END_IF;
   IF #operate.state.ShiftingBottle THEN #operate.machineState := "STATE_SHIFT_BOTTLE"; END_IF;
   IF #operate.state.Stop THEN #operate.machineState := "STATE_STOP"; END_IF;
   IF #operate.state.Reset THEN #operate.machineState := "STATE_RESET"; END_IF;
   IF #operate.state.Error THEN #operate.machineState := "STATE_ERROR"; END_IF;
END_REGION

REGION Network 16: Set machine state OEE
   // 1 = production
   // 2 = planned down
   // 3 = unplanned down
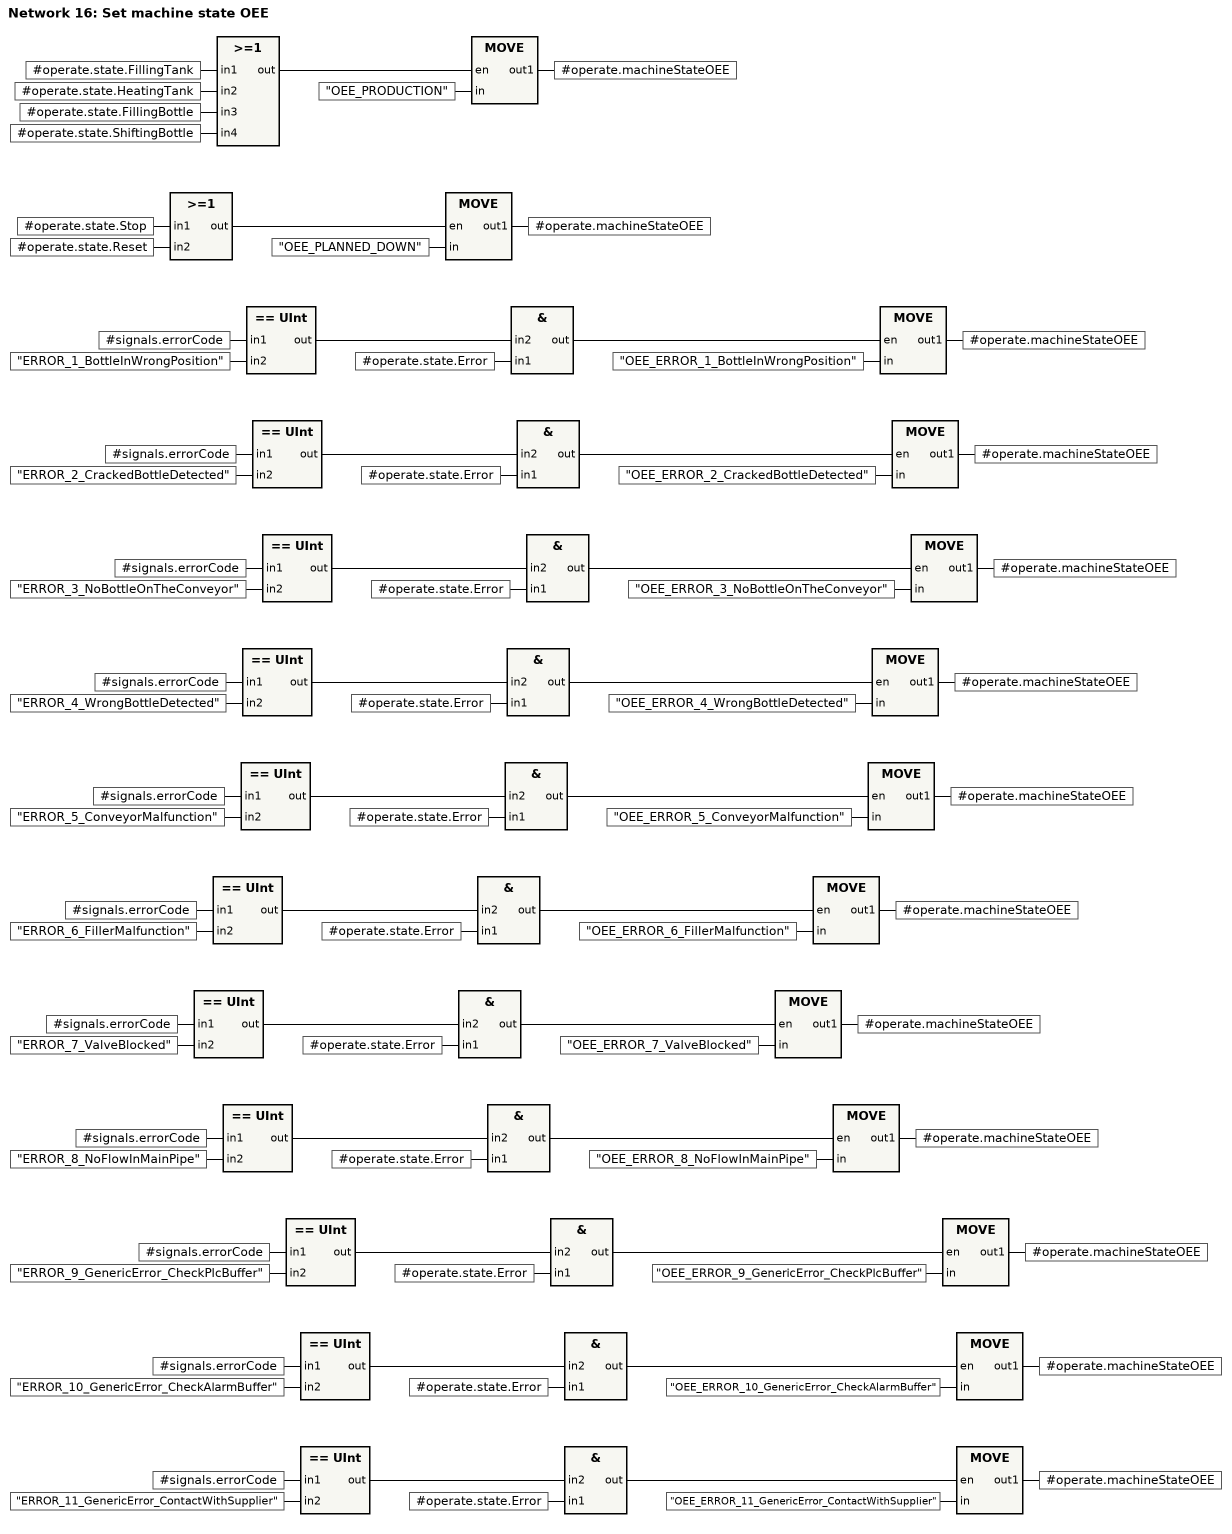
   IF #operate.state.FillingTank OR #operate.state.HeatingTank OR #operate.state.FillingBottle OR #operate.state.ShiftingBottle THEN
       #operate.machineStateOEE := "OEE_PRODUCTION";
   END_IF;
   IF #operate.state.Stop OR #operate.state.Reset THEN
       #operate.machineStateOEE := "OEE_PLANNED_DOWN";
   END_IF;
   IF (#signals.errorCode = "ERROR_1_BottleInWrongPosition") AND #operate.state.Error THEN
       #operate.machineStateOEE := "OEE_ERROR_1_BottleInWrongPosition";
   END_IF;
   IF (#signals.errorCode = "ERROR_2_CrackedBottleDetected") AND #operate.state.Error THEN
       #operate.machineStateOEE := "OEE_ERROR_2_CrackedBottleDetected";
   END_IF;
   IF (#signals.errorCode = "ERROR_3_NoBottleOnTheConveyor") AND #operate.state.Error THEN
       #operate.machineStateOEE := "OEE_ERROR_3_NoBottleOnTheConveyor";
   END_IF;
   IF (#signals.errorCode = "ERROR_4_WrongBottleDetected") AND #operate.state.Error THEN
       #operate.machineStateOEE := "OEE_ERROR_4_WrongBottleDetected";
   END_IF;
   IF (#signals.errorCode = "ERROR_5_ConveyorMalfunction") AND #operate.state.Error THEN
       #operate.machineStateOEE := "OEE_ERROR_5_ConveyorMalfunction";
   END_IF;
   IF (#signals.errorCode = "ERROR_6_FillerMalfunction") AND #operate.state.Error THEN
       #operate.machineStateOEE := "OEE_ERROR_6_FillerMalfunction";
   END_IF;
   IF (#signals.errorCode = "ERROR_7_ValveBlocked") AND #operate.state.Error THEN
       #operate.machineStateOEE := "OEE_ERROR_7_ValveBlocked";
   END_IF;
   IF (#signals.errorCode = "ERROR_8_NoFlowInMainPipe") AND #operate.state.Error THEN
       #operate.machineStateOEE := "OEE_ERROR_8_NoFlowInMainPipe";
   END_IF;
   IF (#signals.errorCode = "ERROR_9_GenericError_CheckPlcBuffer") AND #operate.state.Error THEN
       #operate.machineStateOEE := "OEE_ERROR_9_GenericError_CheckPlcBuffer";
   END_IF;
   IF (#signals.errorCode = "ERROR_10_GenericError_CheckAlarmBuffer") AND #operate.state.Error THEN
       #operate.machineStateOEE := "OEE_ERROR_10_GenericError_CheckAlarmBuffer";
   END_IF;
   IF (#signals.errorCode = "ERROR_11_GenericError_ContactWithSupplier") AND #operate.state.Error THEN
       #operate.machineStateOEE := "OEE_ERROR_11_GenericError_ContactWithSupplier";
   END_IF;
END_REGION

REGION Network 17: Save current operating state for STOP case (only states 1-4)
   // 1 = filling tank
   // 2 = heating tank
   // 3 = filling bottle
   // 4 = shifting bottle
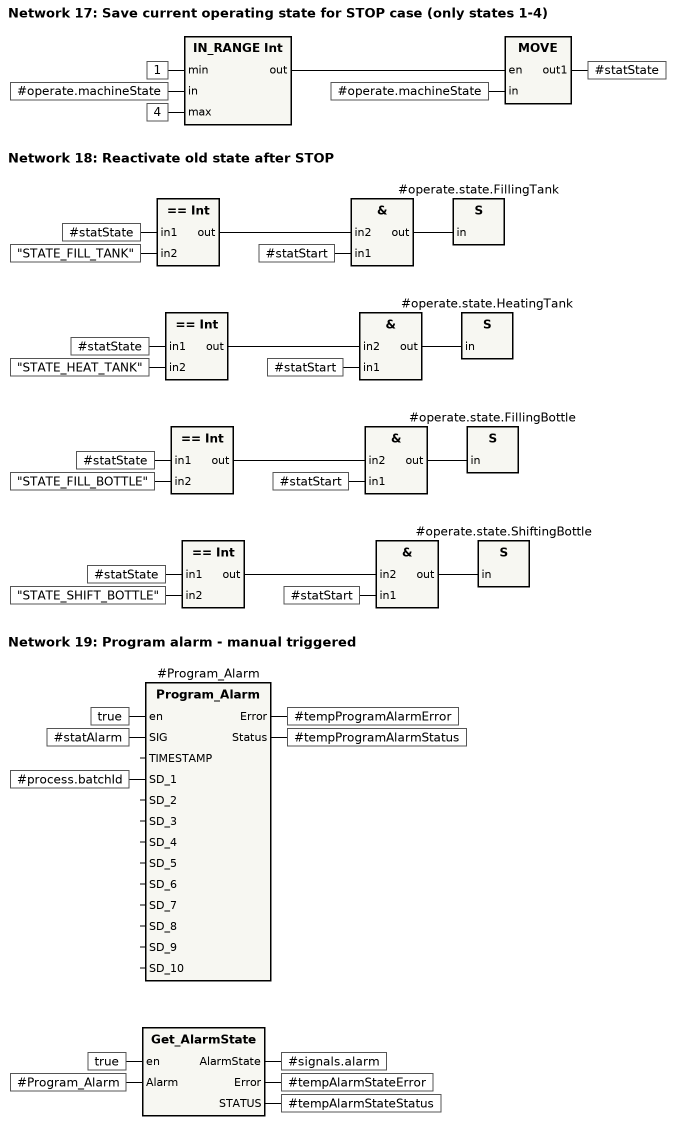
   IF (1 <= #operate.machineState) AND (#operate.machineState <= 4) THEN
       #statState := #operate.machineState;
   END_IF;
END_REGION

REGION Network 18: Reactivate old state after STOP
   // 1 = filling tank
   // 2 = heating tank
   // 3 = filling bottle
   // 4 = shifting bottle
   IF (#statState = "STATE_FILL_TANK") AND #statStart THEN #operate.state.FillingTank := TRUE; END_IF;
   IF (#statState = "STATE_HEAT_TANK") AND #statStart THEN #operate.state.HeatingTank := TRUE; END_IF;
   IF (#statState = "STATE_FILL_BOTTLE") AND #statStart THEN #operate.state.FillingBottle := TRUE; END_IF;
   IF (#statState = "STATE_SHIFT_BOTTLE") AND #statStart THEN #operate.state.ShiftingBottle := TRUE; END_IF;
END_REGION

REGION Network 19: Program alarm - manual triggered
   // no SCL statement known for Get_AlarmState: written as a call
   IF true THEN
       #Program_Alarm(SIG := #statAlarm,   // Program_Alarm
                      SD_1 := #process.batchId,
                      Error => #tempProgramAlarmError,
                      Status => #tempProgramAlarmStatus);
       Get_AlarmState(Alarm := #Program_Alarm,
                      AlarmState => #signals.alarm,
                      Error => #tempAlarmStateError,
                      STATUS => #tempAlarmStateStatus);
   END_IF;
END_REGION

REGION Network 20: Program alarm - out of error code
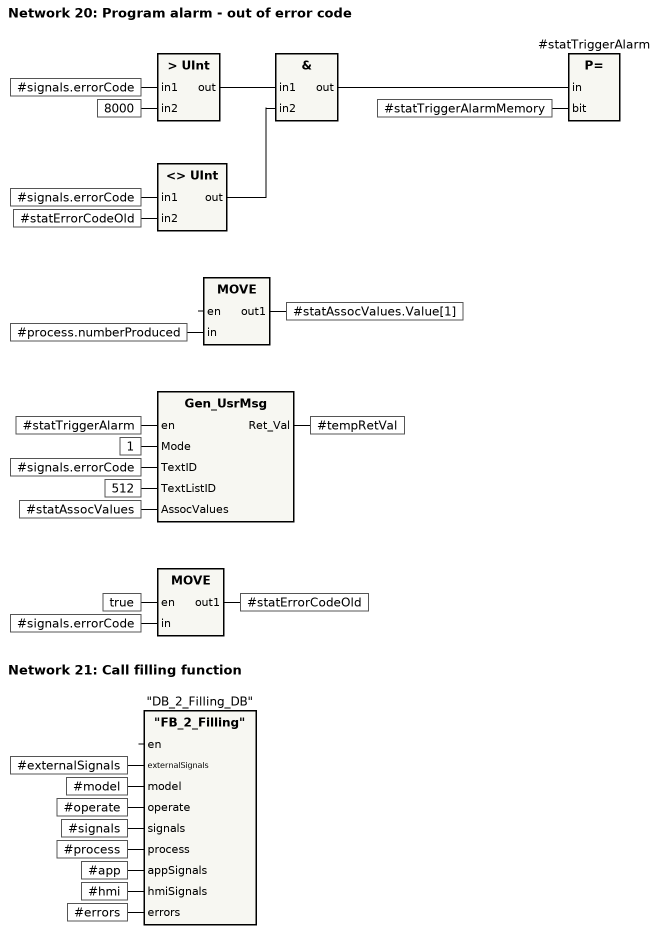
   // no SCL statement known for Gen_UsrMsg: written as a call
   #_w1 := (#signals.errorCode > 8000) AND (#signals.errorCode <> #statErrorCodeOld);
   #statTriggerAlarm := #_w1 AND NOT #statTriggerAlarmMemory;   // rising edge
   #statTriggerAlarmMemory := #_w1;
   #statAssocValues.Value[1] := #process.numberProduced;
   IF #statTriggerAlarm THEN
       #tempRetVal := Gen_UsrMsg(Mode := 1,
                               TextID := #signals.errorCode,
                               TextListID := 512,
                               AssocValues := #statAssocValues);
   END_IF;
   IF true THEN #statErrorCodeOld := #signals.errorCode; END_IF;
END_REGION

REGION Network 21: Call filling function
   "DB_2_Filling_DB"(externalSignals := #externalSignals,   // "FB_2_Filling"
                     model := #model,
                     operate := #operate,
                     signals := #signals,
                     process := #process,
                     appSignals := #app,
                     hmiSignals := #hmi,
                     errors := #errors);
END_REGION
END_FUNCTION_BLOCK

FUNCTION_BLOCK "FB_2_Filling"   // FB3, FBD
TITLE = Filling process
{ S7_Optimized_Access := 'TRUE' }
VERSION : 0.1
   VAR_INPUT
      externalSignals : "typeSignals";   // signals from external model
   END_VAR
   VAR_IN_OUT
      model : "typeModel";   // model parameter
      operate : "typeOperate";   // application operation
      signals : "typeSignals";   // current signals from tank
      process : "typeProcess";   // current process information
      appSignals : "typeApp";
      hmiSignals : "typeHmi";
      errors : "typeError";   // error information
   END_VAR
   VAR
      statShiftingBottle : Bool;
      statShiftingTrigger : Bool;
      statShiftingTimer : Int;
      statHmiBottleLevel : Real;   // parameter for HMI to show current bottle level
      statHmiDoShift : Bool;   // trigger for HMI to shift bottles
      statHmiFaultyBottle : Bool;   // trigger for HMI for faulty bottle
      statBatchIdOld : UDInt := 0;   // helper when batchID changed
      statFillingTankTrigger : Bool;
      statStartCounter : Bool;
      statProducedStart : UDInt;
      statProducedEnd : UDInt;
      statSizeBatchID : USInt;
      statSizeNumberProduced : USInt;
      statStringBatchID : String;
      statStringProductID : String;
   END_VAR
   VAR_TEMP
      tempBottleMaxLevel : Real;
      tempTimerFinished : Bool;
      tempTimeOutput : Time;
      tempCurrentTime : DTL;
      tempTimeRet : Int;
   END_VAR
   VAR_TEMP   // added for the SCL form of the ladder/FBD networks
      _w1 : Bool;
      _w2 : Bool;
   END_VAR
BEGIN

REGION Network 1: Calculation of params
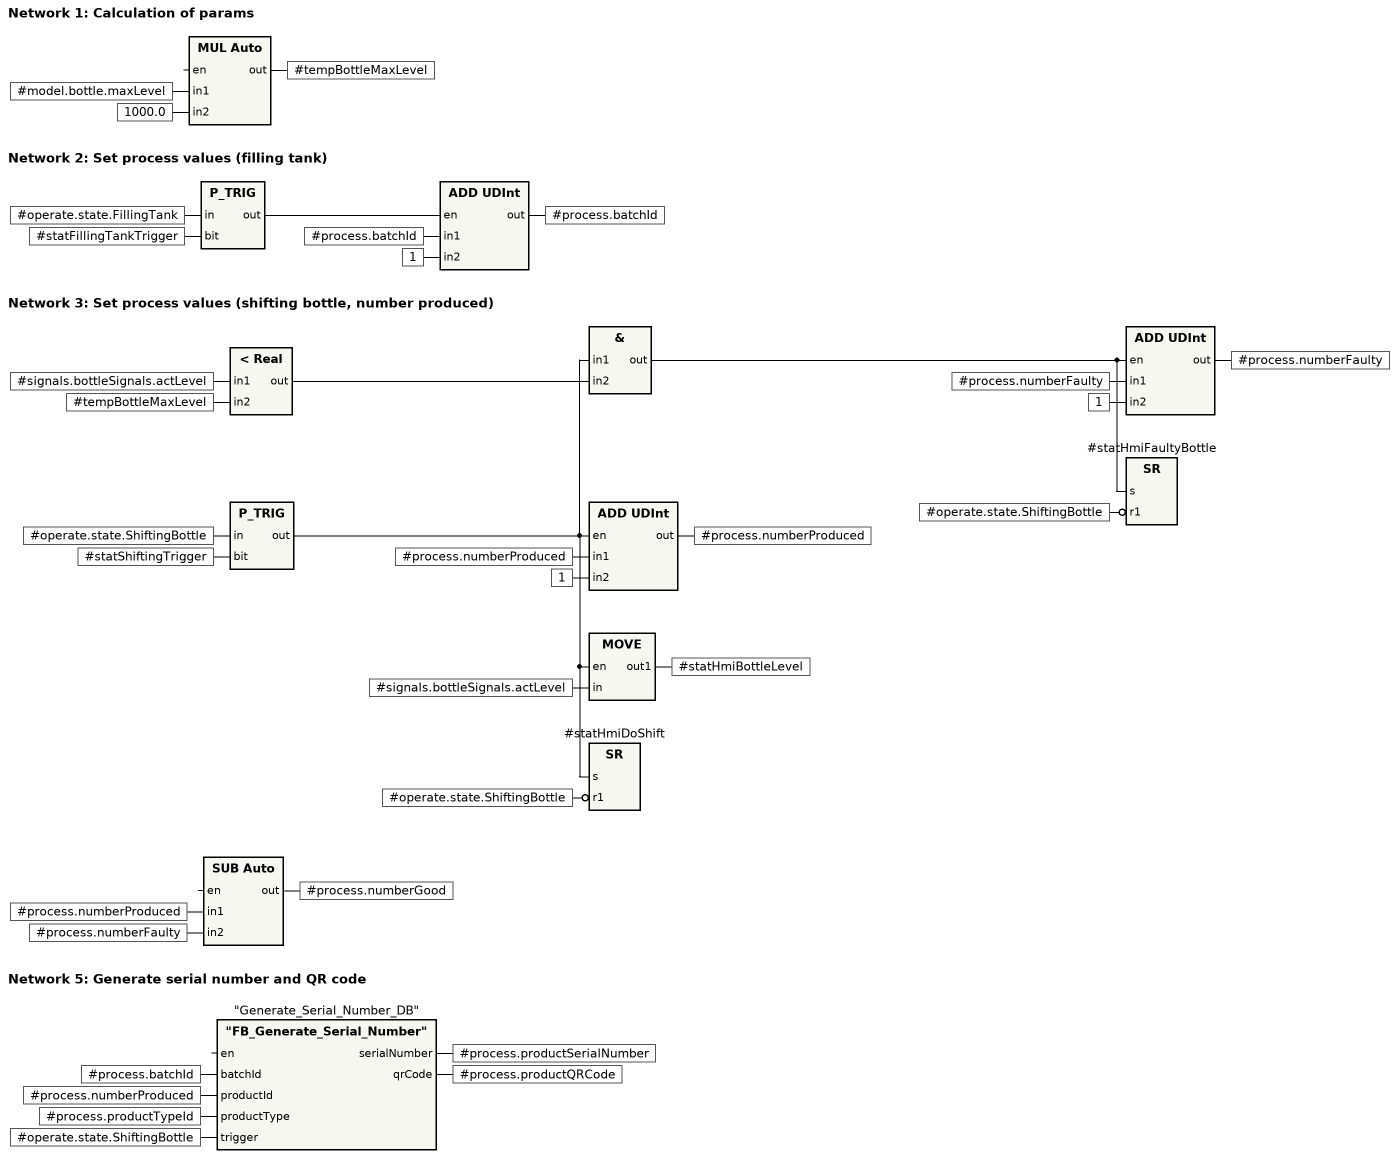
   #tempBottleMaxLevel := #model.bottle.maxLevel * 1000.0;
END_REGION

REGION Network 2: Set process values (filling tank)
   #_w1 := #operate.state.FillingTank AND NOT #statFillingTankTrigger;   // rising edge
   #statFillingTankTrigger := #operate.state.FillingTank;
   IF #_w1 THEN #process.batchId := #process.batchId + 1; END_IF;
END_REGION

REGION Network 3: Set process values (shifting bottle, number produced)
   #_w1 := #operate.state.ShiftingBottle AND NOT #statShiftingTrigger;   // rising edge
   #statShiftingTrigger := #operate.state.ShiftingBottle;
   IF #_w1 THEN #process.numberProduced := #process.numberProduced + 1; END_IF;
   #_w2 := #_w1 AND (#signals.bottleSignals.actLevel < #tempBottleMaxLevel);
   IF #_w2 THEN
       #process.numberFaulty := #process.numberFaulty + 1;
       #statHmiFaultyBottle := TRUE;   // SR flip-flop
   END_IF;
   IF NOT #operate.state.ShiftingBottle THEN #statHmiFaultyBottle := FALSE; END_IF;
   IF #_w1 THEN
       #statHmiBottleLevel := #signals.bottleSignals.actLevel;
       #statHmiDoShift := TRUE;   // SR flip-flop
   END_IF;
   IF NOT #operate.state.ShiftingBottle THEN #statHmiDoShift := FALSE; END_IF;
   #process.numberGood := #process.numberProduced - #process.numberFaulty;
END_REGION

REGION Network 4 (SCL): Set process values (product type ID, name)
   // 1 'Sparkling water'
   // 2 'Medium water'
   // 3 'Still water'
   IF #process.batchId <> #statBatchIdOld THEN

       IF #process.batchId = 1 THEN
           #process.productTypeId := 1;
       ELSE
           IF #process.productTypeId = 3 THEN
               #process.productTypeId := 1;
           ELSE
               #process.productTypeId := #process.productTypeId + 1;
           END_IF;
       END_IF;

       CASE #process.productTypeId OF
           1:  
               #process.productTypeName := 'Sparkling water';
           2:
               #process.productTypeName := 'Medium water';
           3:
               #process.productTypeName := 'Still water';
           ELSE
               #process.productTypeName := 'Undefined';
       END_CASE;

       #statBatchIdOld := #process.batchId;

   END_IF;
END_REGION

REGION Network 5: Generate serial number and QR code
   "Generate_Serial_Number_DB"(batchId := #process.batchId,   // "FB_Generate_Serial_Number"
                           productId := #process.numberProduced,
                           productType := #process.productTypeId,
                           trigger := #operate.state.ShiftingBottle,
                           serialNumber => #process.productSerialNumber,
                           qrCode => #process.productQRCode);
END_REGION

REGION Network 6 (SCL): Calculate production speed (pcs/h)
   // NOT WORKING currently
   // --> fix values as defined in GDB.process.speedActual


   (*

   // get current date
   #tempTimeRet := RD_LOC_T(#tempCurrentTime);  // get local time (DTL)

   // start counting every hour
   IF (#tempCurrentTime.MINUTE = 0 AND #tempCurrentTime.SECOND = 0) THEN
       #statStartCounter := true;
       #statProducedStart := #process.numberProduced;
   END_IF;

   "IEC_Timer_0_DB".TON(IN := #statStartCounter,
                        PT := T#59m_30s,
                        Q => #tempTimerFinished,
                        ET => #tempTimeOutput);

   IF #tempTimerFinished THEN
       #statStartCounter := false;
       #statProducedEnd := #process.numberProduced;
       IF #statProducedEnd > #statProducedStart THEN
           #process.speedActual := #statProducedEnd - #statProducedStart;
       ELSE
           #process.speedActual := 4294967295 - #statProducedStart + #statProducedEnd;
       END_IF;
   END_IF;

   *)
END_REGION

REGION Network 7 (SCL): Generate produt ID (batchID.numberProduced)
   IF #operate.state.ShiftingBottle THEN

       "FC_2_GetStringSizeOfNumber"(number := #process.batchId,
                                    stringSize => #statSizeBatchID);

       "FC_2_GetStringSizeOfNumber"(number := #process.numberProduced,
                                    stringSize => #statSizeNumberProduced);

       VAL_STRG(IN := #process.batchId,
                SIZE := #statSizeBatchID,
                PREC := 0,
                FORMAT := 0,
                P := 1,
                OUT => #statStringBatchID);

       VAL_STRG(IN := #process.numberProduced,
                SIZE := #statSizeNumberProduced,
                PREC := 0,
                FORMAT := 0,
                P := 1,
                OUT => #statStringProductID);

       #process.productId := CONCAT(
                                    IN1 := #statStringBatchID,
                                    IN2 := '.',
                                    IN3 := #statStringProductID
       );
   END_IF;
END_REGION

REGION Network 8 (SCL): Set cycle time
   CASE #operate.machineState OF
       "STATE_FILL_TANK":
           #model.cycleTime := 0.001;
       "STATE_HEAT_TANK":
           #model.cycleTime := 0.001;
       ELSE
           #model.cycleTime := 0.005;
   END_CASE;
END_REGION

REGION Network 9: Simulation (fill tank / heat tank / fill bottle)
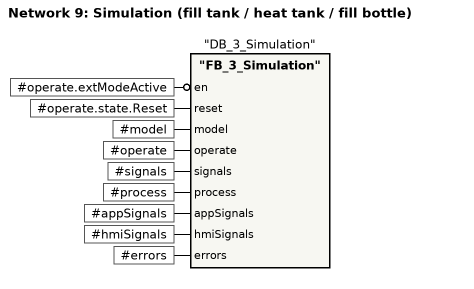
   IF NOT #operate.extModeActive THEN
       "DB_3_Simulation"(reset := #operate.state.Reset,   // "FB_3_Simulation"
                         model := #model,
                         operate := #operate,
                         signals := #signals,
                         process := #process,
                         appSignals := #appSignals,
                         hmiSignals := #hmiSignals,
                         errors := #errors);
   END_IF;
END_REGION

REGION Network 10 (SCL): Reset process parameter
   IF #operate.state.Reset THEN
       #process.batchId := 0;
       #process.numberFaulty := 0;
       #process.numberGood := 0;
       #process.numberProduced := 0;

       #process.productId := '';
       #process.productSerialNumber := '';
       #process.productTypeName := '';
       #process.productQRCode := 0;
       #process.productTypeId := 0;

       #process.speedActual := 0;
       #process.speedTarget := 0;

       #statHmiBottleLevel := 0.0;
       #signals.energySignals.energyConsumptionFillingBottles := 0.0;
       #signals.energySignals.energyConsumptionFillingTank := 0.0;
       #signals.energySignals.energyConsumptionHeatingTank := 0.0;
       #signals.energySignals.waterConsumptionFillingTank := 0.0;
       #signals.energySignals.gasConsumptionHeatingTank := 0.0;

   END_IF;
END_REGION
END_FUNCTION_BLOCK

FUNCTION_BLOCK "FB_3_Simulation"   // FB4, FBD
TITLE = Model Tank Level
{ S7_Optimized_Access := 'TRUE' }
VERSION : 0.1
   VAR_INPUT
      reset : Bool;   // reset tanklevel
      model : "typeModel";   // model parameter
      operate : "typeOperate";   // operate parameter
   END_VAR
   VAR_IN_OUT
      signals : "typeSignals";   // current signals from tank
      process : "typeProcess";   // current process parameters
      appSignals : "typeApp";
      hmiSignals : "typeHmi";
      errors : "typeError";
   END_VAR
   VAR
      "statVinl/min" : Real;   // Vin[l/min]
      "statVinM3/S" : Real;   // Vin [m³/s]
      statInputTanklevel : Real;   // TANK: input tank level for LSim_I [m³]
      statTankLevelSqrt : Real;   // TANK: sqrt of tank level [m³]
      statOutGainSqrt : Real;   // TANK: sqrt of GAIN_SQRT
      statOutGainDiv : Real;   // TANK: divide AB/AT
      statOutGainValue : Real;   // TANK: output gain value
      statVoutSwitch : Real;   // TANK: Vout switch
      statVoutMultiplier : Real;   // TANK: tank level sqrt *output gain value [m³]
      statTankLevel : Real;   // TANK: current level of tank (m³)
      statLiquidMass : Real;   // TANK: liquid mass [kg]
      statLiquidPower : Real;   // TANK: liquid power [N]
      statLiquidPressure_Pa : Real;   // TANK: liquid pressure [Pa]
      instLSim_I_tank : "LSim_I";   // TANK: instance of LSim_I
      statPT1in1 : Real;   // HEAT: input PT1_1
      statPT1out1 : Real;   // HEAT: output PT1_1
      statPT1out2 : Real;   // HEAT: output PT1_2
      instLSim_PT1_1 : "LSim_PT1";   // HEAT: instance PT1 1
      instLSim_PT1_2 : "LSim_PT1";   // HEAT: instance PT1 2
      instLSim_PT1_3 : "LSim_PT1";   // HEAT: instance PT1 3
      instLSim_PT3 : "LSim_PT3";   // HEAT: instance of PT3
      statPT3in : Real;   // HEAT: input value for PT3
      instLSim_I_bottle : "LSim_I";   // BOTTLE: instance of LSim_I
      statBottleLevel : Real;   // BOTTLE: Input bottle level for LSim_I
      statResetHeatingTrigger : Bool;   // trigger for resetting heating
      statResetHeatingMem : Bool;
      statHeatingActive : Bool;   // is set, when heating is active (to 80°C)
      statTriggerResetEnergy : Bool;
      statStopMem : Bool;   // trigger memory for stop
      statShiftingMem : Bool;   // trigger memory for shifting bottle
      statErrorMem : Bool;   // trigger memory for new error
      statResetError : Bool;   // helper bit for error > start workflow
      instTimerError : IEC_TIMER;
      statStart : Bool;   // helper to go in Start state
      statTmLagHeat : Real;   // HEAT: time input for LSim_PT1 -> value per runtime
      statTmLagHeatActive : Real := 1.0;
      statTmLagHeatNotActive : Real := 0.01;
      statTmLagTank : Real := 0.1;   // TANK: time input for Lsim_I
      statTmLagBottle : Real := 0.01;   // BOTTLE: time input for Lsim_I
      statRandomNumberStates : Int;
      statTimerRunning : Bool;
      statRandomState : UDInt;
      instTimerRandomState : IEC_TIMER;
      statTimerDuration : Time;
   END_VAR
   VAR_TEMP
      tempValue : Real;
      tempEnableHeating : Bool;   // enable heating controller
      tempRandomFillingTank : Real;
      tempRandomHeatingTank : Real;
      tempRandomFillingBottle : Real;
      tempRandomFaultyBottles : Int;   // random number for faulty bottle generation
      tempRandomError : Int;   // random number for error code
      tempRandomErrorTrigger : Int;   // random number for error state
      tempStopTrigger : Bool;   // trigger for stop
      tempShiftingTrigger : Bool;   // trigger for shifting bottle
      tempErrorTrigger : Bool;   // trigger for new error
      tempStartTimer : Bool;
   END_VAR
   VAR CONSTANT
      RECALC_VIN : Real := 1.667E-05;   // TANK: 1.667E-05 (1/1000 * 1/60), recalc Vin l/min -> m³/s
      GAIN_SQRT : Real := 19.62;   // TANK: 2*9.81
      GAIN_HEAT : Real := 1.0;   // HEAT: gain value
      ACCELERATION : Real := 9.81;   // gravitational acceleration (a = 9,81 m/s²)
   END_VAR
   VAR_TEMP   // added for the SCL form of the ladder/FBD networks
      _w1 : Bool;
   END_VAR
BEGIN

REGION Network 1: TANK: Vin switch [l/min]
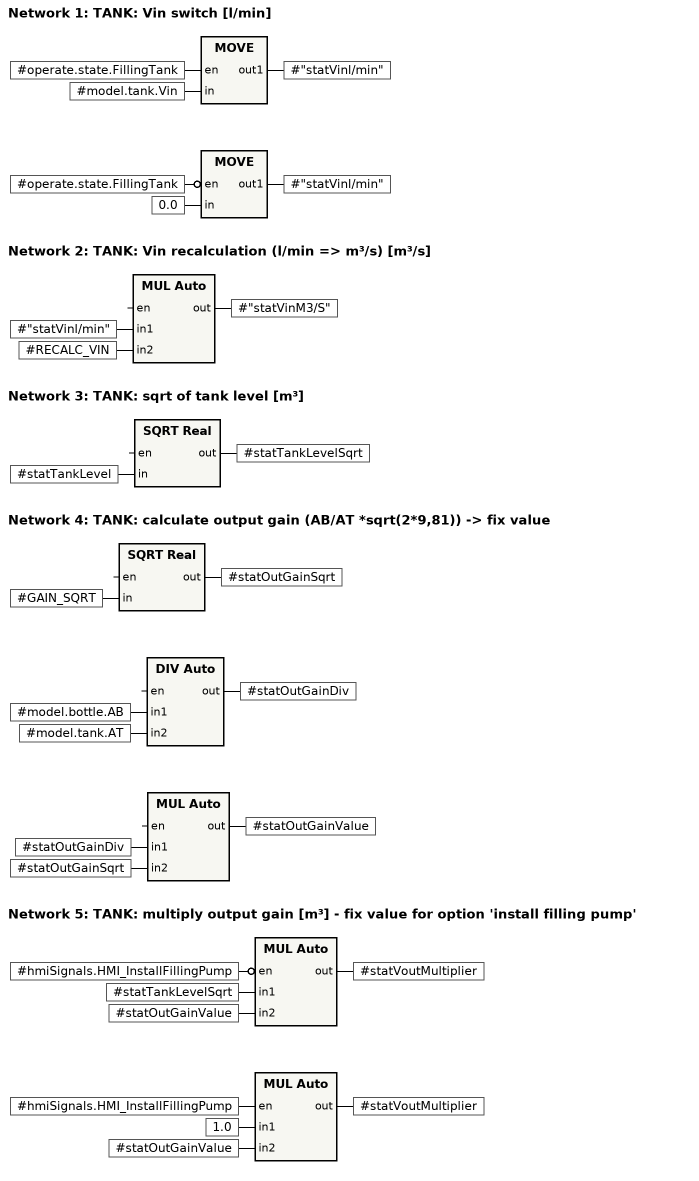
   IF #operate.state.FillingTank THEN #"statVinl/min" := #model.tank.Vin; END_IF;
   IF NOT #operate.state.FillingTank THEN #"statVinl/min" := 0.0; END_IF;
END_REGION

REGION Network 2: TANK: Vin recalculation (l/min => m³/s) [m³/s]
   #"statVinM3/S" := #"statVinl/min" * #RECALC_VIN;
END_REGION

REGION Network 3: TANK: sqrt of tank level [m³]
   #statTankLevelSqrt := SQRT(#statTankLevel);
END_REGION

REGION Network 4: TANK: calculate output gain (AB/AT *sqrt(2*9,81)) -> fix value
   #statOutGainSqrt := SQRT(#GAIN_SQRT);
   #statOutGainDiv := #model.bottle.AB / #model.tank.AT;
   #statOutGainValue := #statOutGainDiv * #statOutGainSqrt;
END_REGION

REGION Network 5: TANK: multiply output gain [m³] - fix value for option 'install filling pump'
   IF NOT #hmiSignals.HMI_InstallFillingPump THEN
       #statVoutMultiplier := #statTankLevelSqrt * #statOutGainValue;
   END_IF;
   IF #hmiSignals.HMI_InstallFillingPump THEN #statVoutMultiplier := 1.0 * #statOutGainValue; END_IF;
END_REGION

REGION Network 6: TANK: Vout switch (input for bottle)
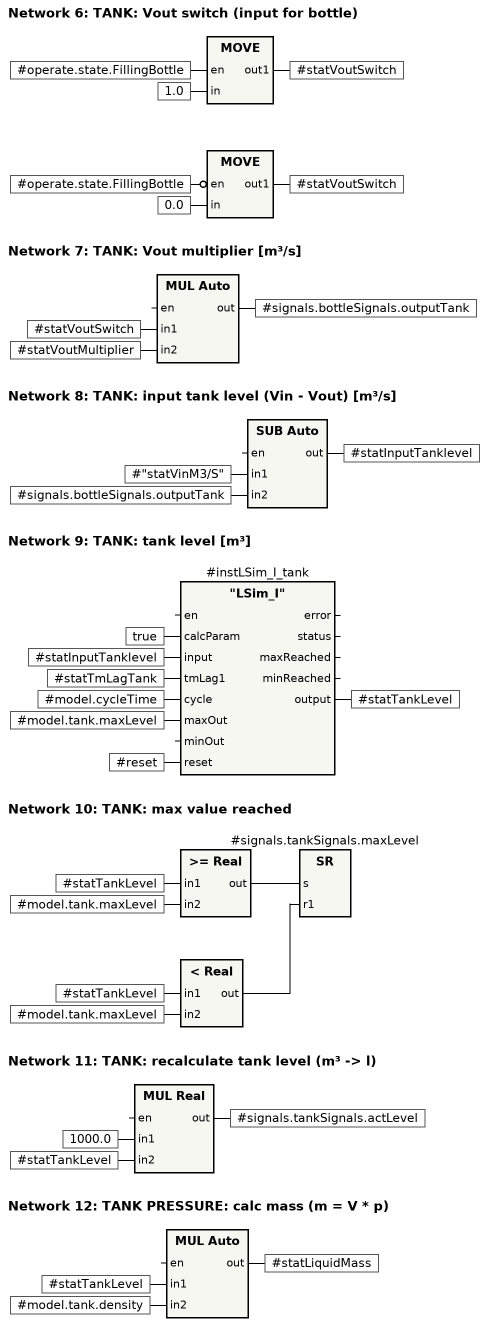
   IF #operate.state.FillingBottle THEN #statVoutSwitch := 1.0; END_IF;
   IF NOT #operate.state.FillingBottle THEN #statVoutSwitch := 0.0; END_IF;
END_REGION

REGION Network 7: TANK: Vout multiplier [m³/s]
   #signals.bottleSignals.outputTank := #statVoutSwitch * #statVoutMultiplier;
END_REGION

REGION Network 8: TANK: input tank level (Vin - Vout) [m³/s]
   #statInputTanklevel := #"statVinM3/S" - #signals.bottleSignals.outputTank;
END_REGION

REGION Network 9: TANK: tank level [m³]
   #instLSim_I_tank(calcParam := true,   // "LSim_I"
                    input := #statInputTanklevel,
                    tmLag1 := #statTmLagTank,
                    cycle := #model.cycleTime,
                    maxOut := #model.tank.maxLevel,
                    reset := #reset,
                    output => #statTankLevel);
END_REGION

REGION Network 10: TANK: max value reached
   IF #statTankLevel >= #model.tank.maxLevel THEN
       #signals.tankSignals.maxLevel := TRUE;   // SR flip-flop
   END_IF;
   IF #statTankLevel < #model.tank.maxLevel THEN #signals.tankSignals.maxLevel := FALSE; END_IF;
END_REGION

REGION Network 11: TANK: recalculate tank level (m³ -> l)
   #signals.tankSignals.actLevel := 1000.0 * #statTankLevel;
END_REGION

REGION Network 12: TANK PRESSURE: calc mass (m = V * p)
   // m = mass [kg]
   // V = volume [m³]
   // p = density [kg/m³]
   #statLiquidMass := #statTankLevel * #model.tank.density;
END_REGION

REGION Network 13: TANK PRESSURE: calc power (F = m * a)
   // F = power [N]
   // m = mass [kg]
   // a = acceleration [m/s²]
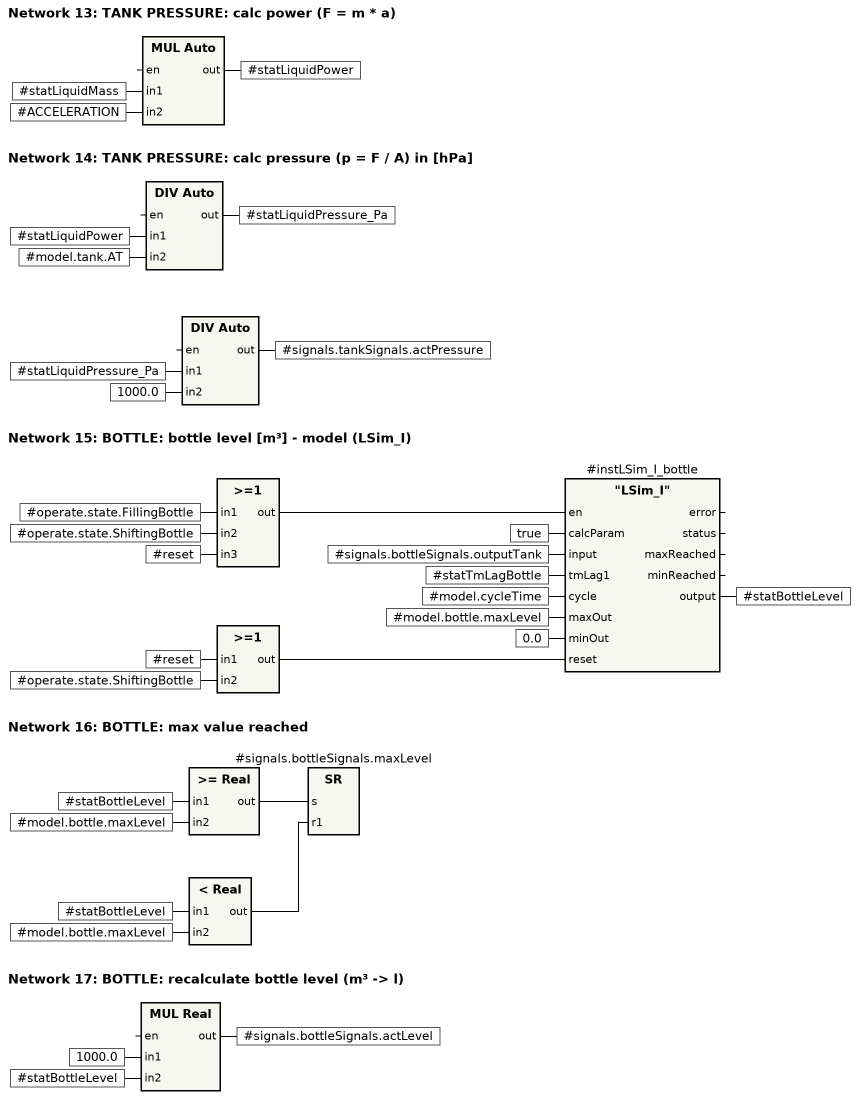
   #statLiquidPower := #statLiquidMass * #ACCELERATION;
END_REGION

REGION Network 14: TANK PRESSURE: calc pressure (p = F / A) in [hPa]
   // p = pressure [Pa]
   // F = power [N]
   // A = surface [m²]
   #statLiquidPressure_Pa := #statLiquidPower / #model.tank.AT;
   #signals.tankSignals.actPressure := #statLiquidPressure_Pa / 1000.0;
END_REGION

REGION Network 15: BOTTLE: bottle level [m³] - model (LSim_I)
   IF #operate.state.FillingBottle OR #operate.state.ShiftingBottle OR #reset THEN
       #instLSim_I_bottle(calcParam := true,   // "LSim_I"
                          input := #signals.bottleSignals.outputTank,
                          tmLag1 := #statTmLagBottle,
                          cycle := #model.cycleTime,
                          maxOut := #model.bottle.maxLevel,
                          minOut := 0.0,
                          reset := #reset OR #operate.state.ShiftingBottle,
                          output => #statBottleLevel);
   END_IF;
END_REGION

REGION Network 16: BOTTLE: max value reached
   IF #statBottleLevel >= #model.bottle.maxLevel THEN
       #signals.bottleSignals.maxLevel := TRUE;   // SR flip-flop
   END_IF;
   IF #statBottleLevel < #model.bottle.maxLevel THEN #signals.bottleSignals.maxLevel := FALSE; END_IF;
END_REGION

REGION Network 17: BOTTLE: recalculate bottle level (m³ -> l)
   #signals.bottleSignals.actLevel := 1000.0 * #statBottleLevel;
END_REGION

REGION Network 18: HEAT: set init values
   // default value (statHeatingActive = false)
   // - temp = 20°C
   // - tmLag = 0.01
   // (set PT1 controller to initial temperature, otherwise PT1 controller would always start at 0°C)
   // 
   // heating phase (statHeatingActive = true)
   // - temp = 80°C
   // - tmLag = 1
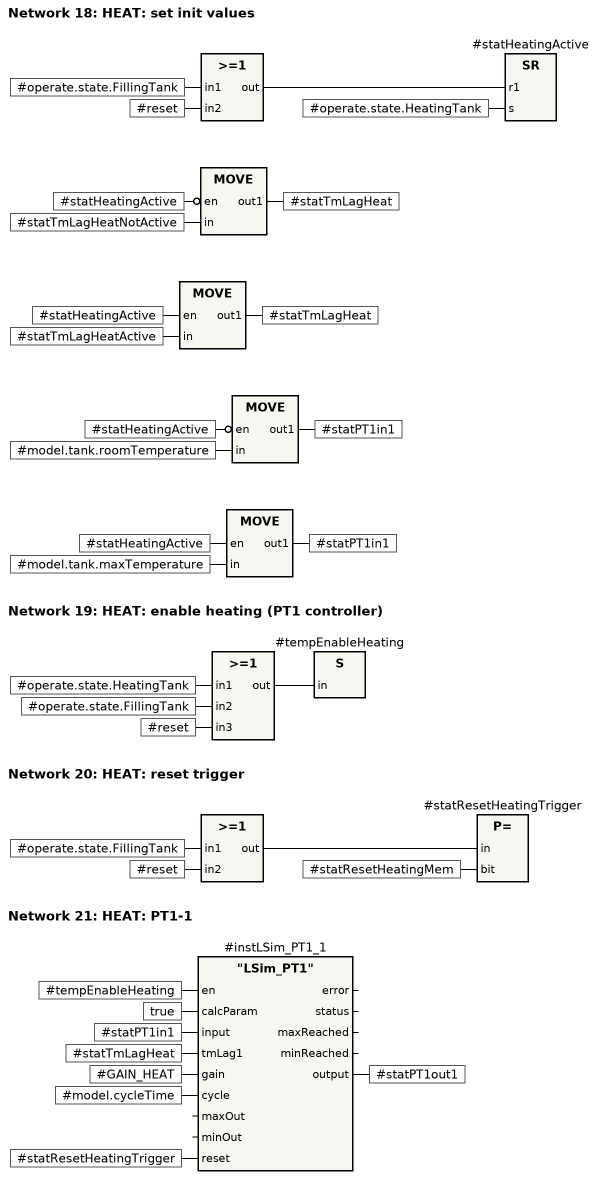
   IF #operate.state.HeatingTank THEN
       #statHeatingActive := TRUE;   // SR flip-flop
   END_IF;
   IF #operate.state.FillingTank OR #reset THEN #statHeatingActive := FALSE; END_IF;
   IF NOT #statHeatingActive THEN #statTmLagHeat := #statTmLagHeatNotActive; END_IF;
   IF #statHeatingActive THEN #statTmLagHeat := #statTmLagHeatActive; END_IF;
   IF NOT #statHeatingActive THEN #statPT1in1 := #model.tank.roomTemperature; END_IF;
   IF #statHeatingActive THEN #statPT1in1 := #model.tank.maxTemperature; END_IF;
END_REGION

REGION Network 19: HEAT: enable heating (PT1 controller)
   IF #operate.state.HeatingTank OR #operate.state.FillingTank OR #reset THEN
       #tempEnableHeating := TRUE;
   END_IF;
END_REGION

REGION Network 20: HEAT: reset trigger
   #_w1 := #operate.state.FillingTank OR #reset;
   #statResetHeatingTrigger := #_w1 AND NOT #statResetHeatingMem;   // rising edge
   #statResetHeatingMem := #_w1;
END_REGION

REGION Network 21: HEAT: PT1-1
   IF #tempEnableHeating THEN
       #instLSim_PT1_1(calcParam := true,   // "LSim_PT1"
                       input := #statPT1in1,
                       tmLag1 := #statTmLagHeat,
                       gain := #GAIN_HEAT,
                       cycle := #model.cycleTime,
                       reset := #statResetHeatingTrigger,
                       output => #statPT1out1);
   END_IF;
END_REGION

REGION Network 22: HEAT: PT1-2
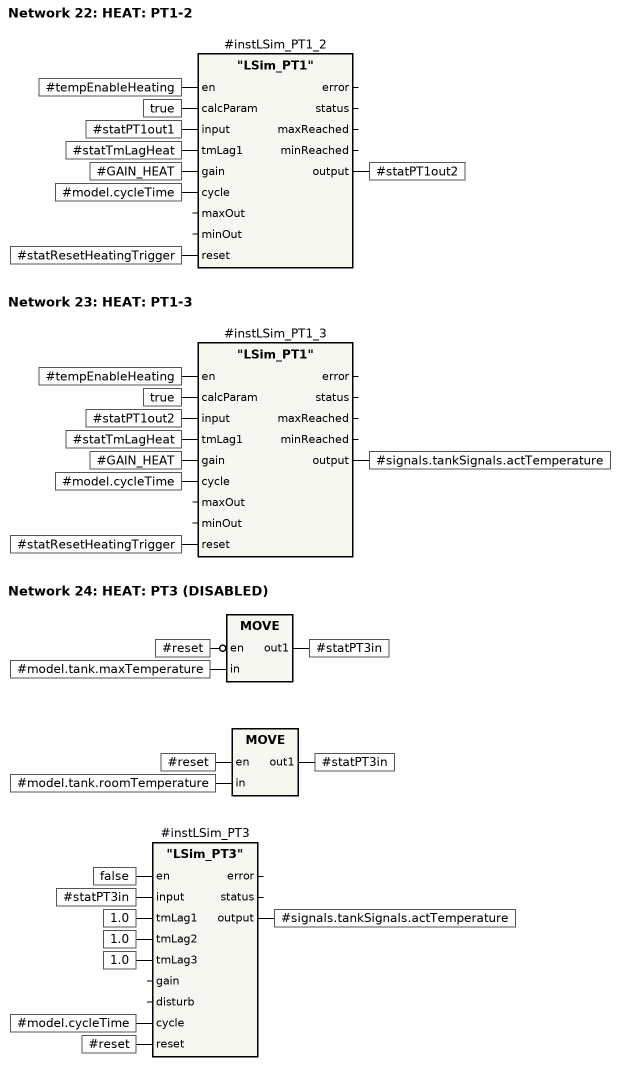
   IF #tempEnableHeating THEN
       #instLSim_PT1_2(calcParam := true,   // "LSim_PT1"
                       input := #statPT1out1,
                       tmLag1 := #statTmLagHeat,
                       gain := #GAIN_HEAT,
                       cycle := #model.cycleTime,
                       reset := #statResetHeatingTrigger,
                       output => #statPT1out2);
   END_IF;
END_REGION

REGION Network 23: HEAT: PT1-3
   IF #tempEnableHeating THEN
       #instLSim_PT1_3(calcParam := true,   // "LSim_PT1"
                       input := #statPT1out2,
                       tmLag1 := #statTmLagHeat,
                       gain := #GAIN_HEAT,
                       cycle := #model.cycleTime,
                       reset := #statResetHeatingTrigger,
                       output => #signals.tankSignals.actTemperature);
   END_IF;
END_REGION

REGION Network 24: HEAT: PT3 (DISABLED)
   IF NOT #reset THEN #statPT3in := #model.tank.maxTemperature; END_IF;
   IF #reset THEN #statPT3in := #model.tank.roomTemperature; END_IF;
   IF false THEN
       #instLSim_PT3(input := #statPT3in,   // "LSim_PT3"
                     tmLag1 := 1.0,
                     tmLag2 := 1.0,
                     tmLag3 := 1.0,
                     cycle := #model.cycleTime,
                     reset := #reset,
                     output => #signals.tankSignals.actTemperature);
   END_IF;
END_REGION

REGION Network 25: HEAT: max value reached
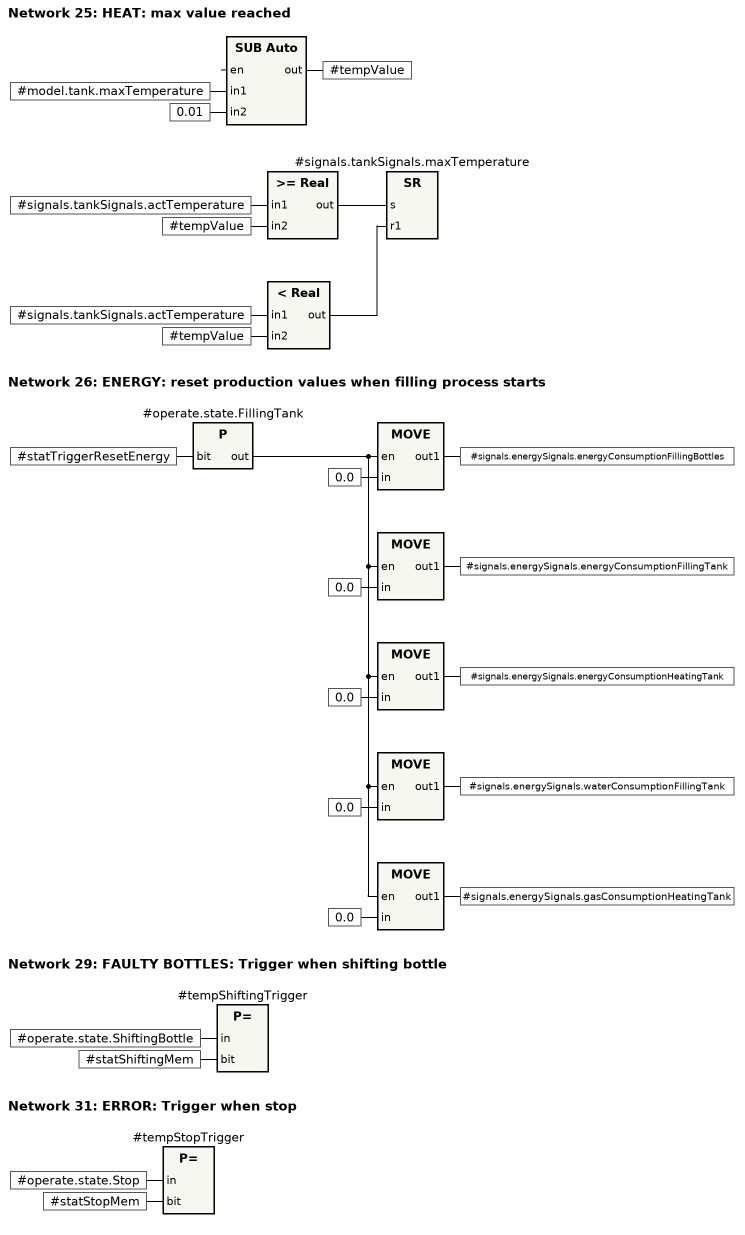
   #tempValue := #model.tank.maxTemperature - 0.01;
   IF #signals.tankSignals.actTemperature >= #tempValue THEN
       #signals.tankSignals.maxTemperature := TRUE;   // SR flip-flop
   END_IF;
   IF #signals.tankSignals.actTemperature < #tempValue THEN
       #signals.tankSignals.maxTemperature := FALSE;
   END_IF;
END_REGION

REGION Network 26: ENERGY: reset production values when filling process starts
   #_w1 := #operate.state.FillingTank AND NOT #statTriggerResetEnergy;   // rising edge of #operate.state.FillingTank
   #statTriggerResetEnergy := #operate.state.FillingTank;
   IF #_w1 THEN
       #signals.energySignals.energyConsumptionFillingBottles := 0.0;
       #signals.energySignals.energyConsumptionFillingTank := 0.0;
       #signals.energySignals.energyConsumptionHeatingTank := 0.0;
       #signals.energySignals.waterConsumptionFillingTank := 0.0;
       #signals.energySignals.gasConsumptionHeatingTank := 0.0;
   END_IF;
END_REGION

REGION Network 27 (SCL): ENERGY: calculate consumption values for filling process
   // generate random values for energy / water / gas consumption
   // energy [Wh] and water [l] consumption during filling tank
   // ----------------------------------------------------------
   IF #operate.state.FillingTank THEN
       "FC_1_Random_Number"(Min := 10,
                       Max := 20,
                       RandomNumber => #tempRandomFillingTank);
       #tempRandomFillingTank := #tempRandomFillingTank / 100;
       #signals.energySignals.energyConsumptionFillingTank := #signals.energySignals.energyConsumptionFillingTank + #tempRandomFillingTank;
       #signals.energySignals.waterConsumptionFillingTank := #signals.tankSignals.actLevel;
   END_IF;

   // energy and gas consumption during heating tank [Wh]
   // ---------------------------------------------------
   IF #operate.state.HeatingTank THEN
       IF #hmiSignals.HMI_RenewHeatingElement THEN
           "FC_1_Random_Number"(Min := 1,
                           Max := 5,
                           RandomNumber => #"tempRandomHeatingTank");
       ELSE
           "FC_1_Random_Number"(Min := 1,
                           Max := 8,
                           RandomNumber => #"tempRandomHeatingTank");
       END_IF;

       #"tempRandomHeatingTank" := #"tempRandomHeatingTank" / 10;
       #signals.energySignals.energyConsumptionHeatingTank := #signals.energySignals.energyConsumptionHeatingTank + #"tempRandomHeatingTank";
       #signals.energySignals.gasConsumptionHeatingTank := #signals.energySignals.gasConsumptionHeatingTank + (#"tempRandomHeatingTank" * 1.5);

   END_IF;

   // energy consumption during filling bottles [Wh]
   // -----------------------------------------------
   IF #operate.state.FillingBottle OR #operate.state.ShiftingBottle THEN
       "FC_1_Random_Number"(Min := 10,
                       Max := 50,
                       RandomNumber => #tempRandomFillingBottle);
       #tempRandomFillingBottle := #tempRandomFillingBottle / 1000;
       #signals.energySignals.energyConsumptionFillingBottles := #signals.energySignals.energyConsumptionFillingBottles + #tempRandomFillingBottle;
   END_IF;
END_REGION

REGION Network 28 (SCL): ENERGY: calculate consumption values per state
   // Standart states: 
   // 1 = powering up
   // 2 = powering down
   // 3 = off
   // 4  = standby
   // 5 = operational
   // 6 = working
   // simulated energy consumption [kWh] for standard machine states (independed from tank process)
   // --------------------------------------------------------------
   "FC_1_Random_Number"(Min := 35,
                        Max := 40,
                        RandomNumber => #statRandomNumberStates);

   // simulate standart states from 1-6
   // ---------------------------------

   // 1 = power up
   // 2 = power donw
   // 3 = off
   // 4 = standby
   // 5 = operational
   // 6 = working

   IF #statTimerRunning = false THEN

       "FC_1_Random_Number"(Min := 1,
                            Max := 500000,
                            RandomNumber => #statRandomState);
   END_IF;

   // State 1-5
   IF #statRandomState >= 1 AND #statRandomState <= 5 THEN

       #signals.energySignalsPerState.stateId := #statRandomState;

       IF #statTimerRunning = false THEN
           #tempStartTimer := true;
       END_IF;

       IF #statRandomState = 4 OR #statRandomState = 5 THEN
           #statTimerDuration := T#20m;
       ELSE
           #statTimerDuration := T#5m;
       END_IF;

       #instTimerRandomState.TP(PT := #statTimerDuration,
                                IN := #tempStartTimer);

       #statTimerRunning := true;

       IF #instTimerRandomState.Q = false THEN
           RESET_TIMER(#instTimerRandomState);
           #statTimerRunning := false;
   END_IF;

       IF #statRandomState = 1 THEN
           // POWER UP
           #signals.energySignalsPerState.energyConsumptionStatePoweringUp := #statRandomNumberStates / 8;

           #signals.energySignalsPerState.energyConsumptionStatePoweringDown := 0;
           #signals.energySignalsPerState.energyConsumptionStateOff := 0;
           #signals.energySignalsPerState.energyConsumptionStateStandby := 0;
           #signals.energySignalsPerState.energyConsumptionStateOperational := 0;
           #signals.energySignalsPerState.energyConsumptionStateWorking := 0;

       ELSIF #statRandomState = 2 THEN
           // POWER DOWN
           #signals.energySignalsPerState.energyConsumptionStatePoweringDown := #statRandomNumberStates / 15;

           #signals.energySignalsPerState.energyConsumptionStatePoweringUp := 0;
           #signals.energySignalsPerState.energyConsumptionStateOff := 0;
           #signals.energySignalsPerState.energyConsumptionStateStandby := 0;
           #signals.energySignalsPerState.energyConsumptionStateOperational := 0;
           #signals.energySignalsPerState.energyConsumptionStateWorking := 0;

       ELSIF #statRandomState = 3 THEN
           // OFF
           #signals.energySignalsPerState.energyConsumptionStateOff := #statRandomNumberStates / 8;

           #signals.energySignalsPerState.energyConsumptionStatePoweringUp := 0;
           #signals.energySignalsPerState.energyConsumptionStatePoweringDown := 0;
           #signals.energySignalsPerState.energyConsumptionStateStandby := 0;
           #signals.energySignalsPerState.energyConsumptionStateOperational := 0;
           #signals.energySignalsPerState.energyConsumptionStateWorking := 0;

       ELSIF #statRandomState = 4 THEN
           // STANDBY
           #signals.energySignalsPerState.energyConsumptionStateStandby := #statRandomNumberStates / 4;

           #signals.energySignalsPerState.energyConsumptionStatePoweringUp := 0;
           #signals.energySignalsPerState.energyConsumptionStatePoweringDown := 0;
           #signals.energySignalsPerState.energyConsumptionStateOff := 0;
           #signals.energySignalsPerState.energyConsumptionStateOperational := 0;
           #signals.energySignalsPerState.energyConsumptionStateWorking := 0;

       ELSIF #statRandomState = 5 THEN
           // OPERATIONAL
           #signals.energySignalsPerState.energyConsumptionStateOperational := #statRandomNumberStates / 2;

           #signals.energySignalsPerState.energyConsumptionStatePoweringUp := 0;
           #signals.energySignalsPerState.energyConsumptionStatePoweringDown := 0;
           #signals.energySignalsPerState.energyConsumptionStateOff := 0;
           #signals.energySignalsPerState.energyConsumptionStateStandby := 0;
           #signals.energySignalsPerState.energyConsumptionStateWorking := 0;

       END_IF;

   ELSE    // WORKING => State 6

       #signals.energySignalsPerState.stateId := 6;
       #signals.energySignalsPerState.energyConsumptionStateWorking := #statRandomNumberStates;

       #signals.energySignalsPerState.energyConsumptionStatePoweringUp := 0;
       #signals.energySignalsPerState.energyConsumptionStatePoweringDown := 0;
       #signals.energySignalsPerState.energyConsumptionStateOff := 0;
       #signals.energySignalsPerState.energyConsumptionStateStandby := 0;
       #signals.energySignalsPerState.energyConsumptionStateOperational := 0;
   END_IF;

   #signals.energySignalsPerState.energyConsumptionStatesTotal :=
   #signals.energySignalsPerState.energyConsumptionStatePoweringUp +
   #signals.energySignalsPerState.energyConsumptionStatePoweringDown +
   #signals.energySignalsPerState.energyConsumptionStateOff +
   #signals.energySignalsPerState.energyConsumptionStateStandby +
   #signals.energySignalsPerState.energyConsumptionStateOperational +
   #signals.energySignalsPerState.energyConsumptionStateWorking;
END_REGION

REGION Network 29: FAULTY BOTTLES: Trigger when shifting bottle
   #tempShiftingTrigger := #operate.state.ShiftingBottle AND NOT #statShiftingMem;   // rising edge
   #statShiftingMem := #operate.state.ShiftingBottle;
END_REGION

REGION Network 30 (SCL): FAULTY BOTTLES: Simulate faulty bottles (generate random number)
   IF #tempShiftingTrigger THEN
       "FC_1_Random_Number"(Min := 0,
                            Max := 10,
                            RandomNumber => #tempRandomFaultyBottles);

       IF #tempRandomFaultyBottles = 1 THEN
           #process.numberFaulty := #process.numberFaulty + 1;
       END_IF;

   END_IF;
END_REGION

REGION Network 31: ERROR: Trigger when stop
   #tempStopTrigger := #operate.state.Stop AND NOT #statStopMem;   // rising edge
   #statStopMem := #operate.state.Stop;
END_REGION

REGION Network 32 (SCL): ERROR: Simulate error
       IF #appSignals.APP_ErrorSimulation THEN

           // random error generation
           IF #tempShiftingTrigger THEN
               "FC_1_Random_Number"(Min := 0,
                               Max := 15000,
                               RandomNumber => #tempRandomErrorTrigger);

               // go into error state
               IF #tempRandomErrorTrigger = 1 THEN
                   #appSignals.APP_Error := true;
               END_IF;

           END_IF;

           // triggered error genertion
           IF #errors.errorTrigger THEN
               #appSignals.APP_Error := true;
           END_IF;


           // if timer finished (negative edge on it's output), go in stop > start again
           "F_TRIG_DB_Error_Finished"(CLK := #instTimerError.Q,
                                      Q => #statResetError);

           // reset error > machine goes automatically into stop
           IF #statResetError THEN
               #appSignals.APP_Error := false;
               #statResetError := false;
               #statStart := true;
           END_IF;

           IF #tempStopTrigger AND #statStart THEN
               #appSignals.APP_Start := true;
               #statStart := false;
           END_IF;

       END_IF;
END_REGION

REGION Network 33: ERROR: Trigger when new error comes in and start timer
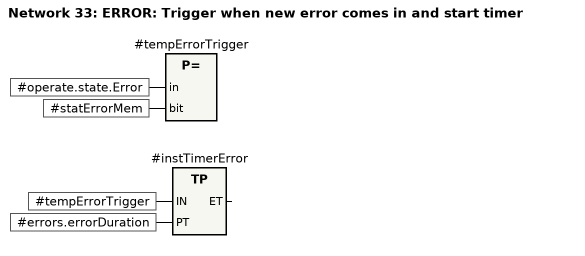
   #tempErrorTrigger := #operate.state.Error AND NOT #statErrorMem;   // rising edge
   #statErrorMem := #operate.state.Error;
   #instTimerError.TP(IN := #tempErrorTrigger, PT := #errors.errorDuration);
END_REGION

REGION Network 34 (SCL): ERROR: Simulate error codes
   // Codes btw. 8001-8011 (8001 = standart HMI error) > see alarm codes
   IF #appSignals.APP_ErrorSimulation THEN

       // generate random error code
       IF #tempErrorTrigger AND (#signals.errorCode = "ERROR_0_NoError") THEN

           "FC_1_Random_Number"(Min := "ERROR_1_BottleInWrongPosition",
                           Max := "ERROR_11_GenericError_ContactWithSupplier",
                           RandomNumber => #tempRandomError);

           #signals.errorCode := INT_TO_UINT(#tempRandomError);

       END_IF;

   END_IF;
END_REGION
END_FUNCTION_BLOCK

FUNCTION_BLOCK "FB_Prodiag"   // FB5, ProDiag
{ S7_Optimized_Access := 'TRUE' }
VERSION : 0.1
   VAR
      PC_Flags : PC_Flags_V2;
      State : SV_FB_State_V2;
   END_VAR
   VAR_TEMP
      t_TempSvStateUDT : SV_State_V2;
      t_TempAlarmInstance : <type 200004f>;
      t_TempAsocValue1 : Variant;
      t_TempAsocValue2 : Variant;
      t_TempAsocValue3 : Variant;
   END_VAR
BEGIN
END_FUNCTION_BLOCK

FUNCTION_BLOCK "FB_4_CIP_Simulation"   // FB6, FBD
{ S7_Optimized_Access := 'TRUE' }
VERSION : 0.1
   VAR_OUTPUT
      startCip : Bool;   // start CIP S7 graph sequence
      stopCip : Bool;   // stop CIP S7 graph sequence
   END_VAR
   VAR_IN_OUT
      cip : "typeCIP";
   END_VAR
   VAR
      statMemoryActive : Bool;
      statSystemTime : DTL;
      statTemperature : Real;
      statStartStep1 : Bool;
      statStartStep2 : Bool;
      statStartStep3 : Bool;
      statStartStep4 : Bool;
      statConcentration : Real;
   END_VAR
   VAR_TEMP
      tempRet : Int;
      tempRandomConcentration : Real;
      tempRandomFlowrate : Real;
      tempStartInit : Bool;
      tempStartStep1 : Bool;
      tempStartStep2 : Bool;
      tempStartStep3 : Bool;
      tempStartStep4 : Bool;
      tempEnd : Bool;
      tempCurrentDate : DTL;   // current date
      tempDateDiff : Time;   // difference bzw. start and current time
      tempStartTime : Time;   // start time
      tempCurrentTOD : Time_Of_Day;   // current time-of-day
      tempCurrentTime : Time;   // current time
      tempStartDate : DTL;   // start date
      tempTimeOut : Time;   // TON timer output
   END_VAR
BEGIN

REGION Network 1 (SCL): CIP simulation
   // start CIP
   // ----------

   // get current date
   #tempRet := RD_LOC_T(#tempCurrentDate);     // get local time (DTL)

   // START with configured #cipStartTime
   // ------------------------------------
   (*
   // get start date (DTL)
   #tempStartDate := TOD_TO_DTL(#cip.cipStartTime);

   // Start CIP process
   IF (#tempCurrentDate.HOUR = #tempStartDate.HOUR) AND (#tempCurrentDate.MINUTE = #tempStartDate.MINUTE) AND (#tempCurrentDate.SECOND = #tempStartDate.SECOND) THEN
       #cip.cipActive := true;
   END_IF;
   *)

   // START every 1 hour
   // -------------------

   // Start CIP process
   IF (#tempCurrentDate.MINUTE = 0 AND #tempCurrentDate.SECOND = 0) THEN
       #cip.cipActive := true;
   END_IF;


   IF #cip.cipActive = false THEN
       #cip.cipProcess := ''; 
       #cip.cipStep := '';
       #cip.cipTemperature := 0;
       #cip.cipConcentration := 0;
       #cip.cipFlowrate := 0;
       #cip.cipStep1 := false;
       #cip.cipStep2 := false;
       #cip.cipStep3 := false;
       #cip.cipStep4 := false;
   END_IF;

   IF #cip.cipActive = true THEN
       #cip.cipProcess := 'Full wash';
   END_IF;

   // INIT Step (1 second)
   "R_TRIG_CIP_Step1"(CLK := #cip.cipActive, Q => #tempStartInit);

   IF #tempStartInit THEN
       #cip.cipId := #cip.cipId + 1;
   END_IF;

   // start S7 graph (official input of graph block)
   #startCip := #tempStartInit;

   // STEP1 (after 1 second)
   "IEC_Timer_CIP_Init".TON(IN:=#cip.cipActive,
                            PT:=T#1s,
                            Q=>#tempStartStep1,
                            ET=>#tempTimeOut);

   IF #tempStartStep1 THEN
       #cip.cipStep4 := false;
       #cip.cipStep1 := true;
       #cip.cipStep := 'pre-rinse';
       #cip.cipTemperature := 125.0;
   END_IF;

   // STEP 2 (after 6 minutes)
   "IEC_Timer_CIP_Step2".TON(IN := #cip.cipActive,
                         PT := T#6m,
                         Q => #tempStartStep2,
                         ET => #tempTimeOut);

   IF #tempStartStep2 THEN
       #cip.cipStep1 := false;
       #cip.cipStep2 := true;

       #cip.cipStep := 'alkali-wash';
       #cip.cipTemperature := 227.0;
       #cip.cipConcentration := 340.0;
   END_IF;

   // STEP 3 (after 22 minutes)
   "IEC_Timer_CIP_Step3".TON(IN := #cip.cipActive,
                             PT := T#22m,
                             Q => #tempStartStep3,
                             ET => #tempTimeOut);

   IF #tempStartStep3 THEN
       #cip.cipStep2 := false;
       #cip.cipStep3 := true;

       #cip.cipStep := 'acid-wash';
       #cip.cipTemperature := 840.0;
       #cip.cipConcentration := 2013.0;
   END_IF;

   // STEP 4 (after 44 minutes)
   "IEC_Timer_CIP_Step4".TON(IN := #cip.cipActive,
                             PT := T#44m,
                             Q => #tempStartStep4,
                             ET => #tempTimeOut);
   IF #tempStartStep4 THEN
       #cip.cipStep3 := false;
       #cip.cipStep4 := true;

       #cip.cipStep := 'final-rinse';
       #cip.cipTemperature := 347.0;
       #cip.cipConcentration := 1830.0;
   END_IF;

   // END
   "IEC_Timer_CIP_End".TON(IN := #cip.cipActive,
                           PT := T#58m,
                           Q => #tempEnd,
                           ET => #tempTimeOut);

   IF #tempEnd THEN
       #cip.cipActive := false;
   END_IF;

   // stop s7 graph
   #stopCip := #tempEnd OR NOT #cip.cipActive;
END_REGION
END_FUNCTION_BLOCK

FUNCTION_BLOCK "FB_5_CIP_Simulation_Graph"   // FB7, GRAPH_PLUS
{ S7_Optimized_Access := 'TRUE' }
VERSION : 0.1
   VAR_INPUT
      OFF_SQ : Bool := false;   // Turn sequence off
      INIT_SQ : Bool := false;   // Set sequence to initial state
      ACK_EF : Bool := false;   // Acknowledge all errors and faults
      S_PREV : Bool := false;   // Output previous step in parameter S_NO
      S_NEXT : Bool := false;   // Indicate next step in parameter S_NO
      SW_AUTO : Bool := false;   // Automatic mode
      SW_TAP : Bool := false;   // Semiautomatic/switch with transition
      SW_TOP : Bool := false;   // Semiautomatic/ignore transition
      SW_MAN : Bool := false;   // Manual mode
      S_SEL : Int := 0;   // Select step to be output to S_NO
      S_ON : Bool := false;   // Activate step indicated in S_NO
      S_OFF : Bool := false;   // Disable step indicated in S_NO
      T_PUSH : Bool := false;   // Enable transition to switch in semi automatic mode
   END_VAR
   VAR_OUTPUT
      S_NO : Int := 0;   // Step number
      S_MORE : Bool := false;   // More steps are available and can be shown in S_NO
      S_ACTIVE : Bool := false;   // Step indicated in S_NO is active
      ERR_FLT : Bool := false;   // Interlock or supervision group error
      AUTO_ON : Bool := false;   // Automatic mode is active
      TAP_ON : Bool := false;   // Semiautomatic mode/step with transition enabled
      TOP_ON : Bool := false;   // Semiautomatic mode/ignore transition enabled
      MAN_ON : Bool := false;   // Manual mode is active
   END_VAR
   VAR_IN_OUT
      cip : "typeCIP";
      stepInitial : Bool;   // Initial step is active
      step1Active : Bool;   // Step 1 is active
      step2Active : Bool;   // Step 2 is active
      step3Active : Bool;   // Step 3 is active
      step4Active : Bool;   // Step 4 is active
   END_VAR
   VAR
      statTemperature : Real;
      statConcentration : Real;
      statAbnomaly : Real;
      HMI_INFO : Array[0..8] of UInt;
      IF_PAR : G7_IfParPlus_V6;
      RT_DATA : G7_RTDataPlus_V6;   // Internal data area
      "Start step 1" : G7_TransitionPlus_V6;   // Transition structure
      "Start step 2" : G7_TransitionPlus_V6;   // Transition structure
      "Start step 3" : G7_TransitionPlus_V6;   // Transition structure
      "Start step 4" : G7_TransitionPlus_V6;   // Transition structure
      End : G7_TransitionPlus_V6;   // Transition structure
      Trans8 : G7_TransitionPlus_V6;   // Transition structure
      "Initial step" : G7_StepPlus_V6;   // Step structure
      "Step1: pre-rinse" : G7_StepPlus_V6;   // Step structure
      "Step2: alkali-wash" : G7_StepPlus_V6;   // Step structure
      "Step3: acid-wash" : G7_StepPlus_V6;   // Step structure
      "Step4: final-rinse" : G7_StepPlus_V6;   // Step structure
      Reset : G7_StepPlus_V6;   // Step structure
      SINI : Array[0..1] of USInt;
      LSTT : Array[0..5] of USInt;
      ATAJ : Array[0..5] of USInt;
      ATAB : Array[0..5] of USInt;
      PSTT : Array[0..5] of USInt;
      NSTT : Array[0..5] of USInt;
      ASSJ : Array[0..5] of USInt;
      ASSB : Array[0..5] of USInt;
      PTTS : Array[0..5] of USInt;
      NTTS : Array[0..5] of USInt;
      SW_SQTS : Array[0..5] of USInt;
      SWITCH : Array[0..0] of USInt;
      TVX : Array[0..1] of USInt;
      TTX : Array[0..1] of USInt;
      TSX : Array[0..1] of USInt;
      S00X : Array[0..1] of USInt;
      SOFFX : Array[0..1] of USInt;
      SONX : Array[0..1] of USInt;
      SAX : Array[0..1] of USInt;
      SERRX : Array[0..6] of USInt;
      SMX : Array[0..6] of USInt;
      S0X : Array[0..6] of USInt;
      S1X : Array[0..6] of USInt;
      IL_ALARM_INST : Diag_Alarm;
      SUP_ALARM_INST : Diag_Alarm;
      STEP_TIME_ALARM_INST : Diag_Alarm;
      IEC_TIMER_INST : IEC_TIMER;
      TRANSACTION_FLAG : Bool := false;
   END_VAR
   VAR_TEMP
      tempRet : Int;
      tempRandomFlowrate : Int;
      tempRandomAbnomaly : Real;
   END_VAR
   // SINI[0] := 2;
   // LSTT[0] := 255;
   // LSTT[1] := 255;
   // LSTT[2] := 255;
   // LSTT[3] := 255;
   // LSTT[4] := 255;
   // ATAJ[1] := 1;
   // ATAJ[2] := 2;
   // ATAJ[3] := 3;
   // ATAJ[4] := 4;
   // ATAB[1] := 1;
   // ATAB[2] := 2;
   // ATAB[3] := 3;
   // ATAB[4] := 4;
   // PSTT[1] := 1;
   // PSTT[2] := 2;
   // PSTT[3] := 3;
   // PSTT[4] := 4;
   // NSTT[0] := 1;
   // NSTT[1] := 2;
   // NSTT[2] := 3;
   // NSTT[3] := 4;
   // NSTT[4] := 5;
   // ASSJ[1] := 1;
   // ASSJ[2] := 2;
   // ASSJ[3] := 3;
   // ASSJ[4] := 4;
   // ASSB[1] := 1;
   // ASSB[2] := 2;
   // ASSB[3] := 3;
   // ASSB[4] := 4;
   // PTTS[0] := 255;
   // PTTS[2] := 1;
   // PTTS[3] := 2;
   // PTTS[4] := 3;
   // NTTS[1] := 1;
   // NTTS[2] := 2;
   // NTTS[3] := 3;
   // NTTS[4] := 4;
   // TVX[0] := 16#1;
   // TTX[0] := 16#1;
   // TSX[0] := 16#1;
   // S00X[0] := 16#1;
   // SOFFX[0] := 16#1;
   // SONX[0] := 16#1;
   // SAX[0] := 16#1;
   // SERRX[0] := 16#1;
   // SMX[0] := 16#1;
   // S0X[0] := 16#1;
   // S1X[0] := 16#1;
   // ATAB[5] := 5;
   // ATAJ[5] := 5;
   // LSTT[5] := 255;
   // PSTT[5] := 5;
   // NSTT[5] := 255;
   // ASSJ[5] := 5;
   // ASSB[5] := 5;
   // PTTS[5] := 4;
   // NTTS[5] := 5;
BEGIN
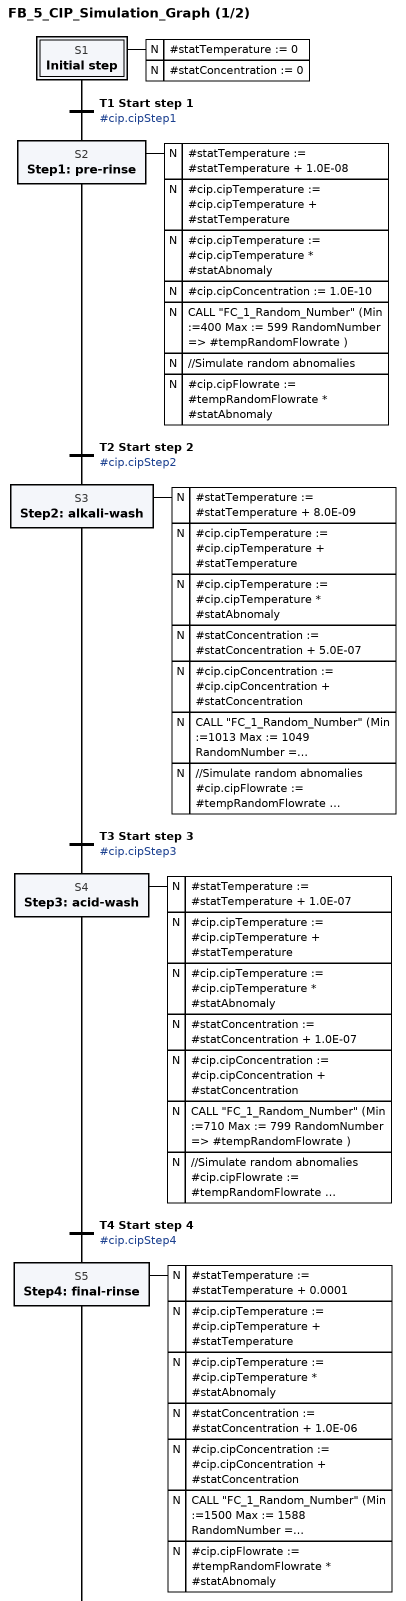
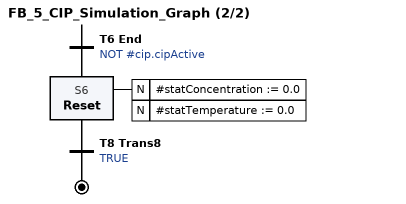
   // permanent pre-instructions
   NETWORK 1
   TITLE = Simulate random abnomalies
      "FC_1_Random_Number"(Min := 70, Max := 100, RandomNumber => #tempRandomAbnomaly);
      #statAbnomaly := #tempRandomAbnomaly / 100.0;

   // sequencer 1
   INITIAL_STEP "Initial step":   // S1, max time T#10S, warning time T#7S
              N    #statTemperature := 0
              N    #statConcentration := 0
   END_STEP
   TRANSITION "Start step 1" FROM "Initial step" TO "Step1: pre-rinse"   // T1
      := #cip.cipStep1;
   END_TRANSITION
   STEP "Step1: pre-rinse":   // S2, max time T#10S, warning time T#7S
              N    #statTemperature := #statTemperature + 1.0E-08
              N    #cip.cipTemperature := #cip.cipTemperature + #statTemperature
              N    #cip.cipTemperature := #cip.cipTemperature * #statAbnomaly
              N    #cip.cipConcentration := 1.0E-10
              N    CALL "FC_1_Random_Number"
                   (Min :=400
                   Max := 599
                   RandomNumber => #tempRandomFlowrate
                   )
                   //Simulate random abnomalies
              N    #cip.cipFlowrate := #tempRandomFlowrate * #statAbnomaly
   END_STEP
   TRANSITION "Start step 2" FROM "Step1: pre-rinse" TO "Step2: alkali-wash"   // T2
      := #cip.cipStep2;
   END_TRANSITION
   STEP "Step2: alkali-wash":   // S3, max time T#10S, warning time T#7S
              N    #statTemperature := #statTemperature + 8.0E-09
              N    #cip.cipTemperature := #cip.cipTemperature + #statTemperature
              N    #cip.cipTemperature := #cip.cipTemperature * #statAbnomaly
              N    #statConcentration := #statConcentration + 5.0E-07
              N    #cip.cipConcentration := #cip.cipConcentration + #statConcentration
              N    CALL "FC_1_Random_Number"
                   (Min :=1013
                   Max := 1049
                   RandomNumber => #tempRandomFlowrate
                   )
              N    //Simulate random abnomalies
                   #cip.cipFlowrate := #tempRandomFlowrate * #statAbnomaly
   END_STEP
   TRANSITION "Start step 3" FROM "Step2: alkali-wash" TO "Step3: acid-wash"   // T3
      := #cip.cipStep3;
   END_TRANSITION
   STEP "Step3: acid-wash":   // S4, max time T#10S, warning time T#7S
              N    #statTemperature := #statTemperature + 1.0E-07
              N    #cip.cipTemperature := #cip.cipTemperature + #statTemperature
              N    #cip.cipTemperature := #cip.cipTemperature * #statAbnomaly
              N    #statConcentration := #statConcentration + 1.0E-07
              N    #cip.cipConcentration := #cip.cipConcentration + #statConcentration
              N    CALL "FC_1_Random_Number"
                   (Min :=710
                   Max := 799
                   RandomNumber => #tempRandomFlowrate
                   )
              N    //Simulate random abnomalies
                   #cip.cipFlowrate := #tempRandomFlowrate * #statAbnomaly
   END_STEP
   TRANSITION "Start step 4" FROM "Step3: acid-wash" TO "Step4: final-rinse"   // T4
      := #cip.cipStep4;
   END_TRANSITION
   STEP "Step4: final-rinse":   // S5, max time T#10S, warning time T#7S
              N    #statTemperature := #statTemperature + 0.0001
              N    #cip.cipTemperature := #cip.cipTemperature + #statTemperature
              N    #cip.cipTemperature := #cip.cipTemperature * #statAbnomaly
              N    #statConcentration := #statConcentration + 1.0E-06
              N    #cip.cipConcentration := #cip.cipConcentration + #statConcentration
              N    CALL "FC_1_Random_Number"
                   (Min :=1500
                   Max := 1588
                   RandomNumber => #tempRandomFlowrate
                   )
              N    #cip.cipFlowrate := #tempRandomFlowrate * #statAbnomaly
   END_STEP
   TRANSITION End FROM "Step4: final-rinse" TO Reset   // T6
      := NOT #cip.cipActive;
   END_TRANSITION
   STEP Reset:   // S6, max time T#10S, warning time T#7S
              N    #statConcentration := 0.0
              N    #statTemperature := 0.0
   END_STEP
   TRANSITION Trans8 FROM Reset TO END   // T8
      := TRUE;
   END_TRANSITION

   // permanent post-instructions
   NETWORK 1
   TITLE = transfer states to output
      #step1Active := #"Step1: pre-rinse".X;
      #step2Active := #"Step2: alkali-wash".X;
      #step3Active := #"Step3: acid-wash".X;
      #step4Active := #"Step4: final-rinse".X;
      #stepInitial := #"Initial step".X;
END_FUNCTION_BLOCK

FUNCTION_BLOCK "LSim_PT1"   // FB50, SCL
{ S7_Optimized_Access := 'TRUE' }
VERSION : 2.01
   VAR_INPUT
      calcParam : Bool;   // recalculate with new parameters
      input : Real;   // input signal
      tmLag1 : Real := 1.0;   // time constant T1 [sec]
      gain : Real := 1.0;   // gain factor
      cycle : Real := 0.1;   // cyclic time [sec]
      maxOut : Real := 100.0;   // max. output limit
      minOut : Real;   // min. output limit
      reset : Bool;   // resets all relevant parameters to ‘0’ including the output
   END_VAR
   VAR_OUTPUT
      error : Bool;   // error (#tmLag1 <= 0)
      status : Word;   // status (if #tmLag1 <= 0 then status = 16#8001)
      maxReached : Bool;   // output has reached max. limit
      minReached : Bool;   // output has reached min. limit
      output : Real;   // output signal (if #error = FALSE)
   END_VAR
   VAR
      statRf1 : Real;
      statRe1 : Real;
      statOverfirst : Bool;
      statOutput : Real;
   END_VAR
BEGIN
   //=============================================================================
   //SIEMENS AG
   //(c)Copyright 2017 All Rights Reserved
   //-----------------------------------------------------------------------------
   //Library:       Library for Controlled System Simulation
   //Tested with:   S7-1500 FW V2.0 / S7-1200 FW V4.2
   //Engineering:   STEP 7 V14 Upd2 (TIA Portal)
   //Restrictions:  Cyclic interrupt
   //Requirements:  memory card needed for S7-1500
   //Functionality: Simulation of a PT1-System
   //
   //              gain
   //  F(p) = ---------------
   //          tmLag1 * p + 1
   //          
   //  Call the simulation in a cyclic interrupt with
   //  cyclic interrupt time at least = tmLag1/10!
   //-----------------------------------------------------------------------------
   //Change log table:
   //Version  Date       Expert in charge                Changes applied
   //02.00.00 03.02.2016 Siemens Industry Online Support Release (STEP 7 V13 SP1)
   //02.00.01 02.03.2017 Siemens Industry Online Support Release (STEP 7 V14)
   //=============================================================================
   // check parameter
   IF #tmLag1 <= 0 THEN
     #error := TRUE;
     #status := W#16#8001;     // Parameter Error
     #statOutput := 0;
     #output := 0;
     RETURN;
   ELSE
     #error := FALSE;
     #status := W#16#0000;     // no error
   END_IF;

   IF #calcParam = True OR NOT #statOverfirst THEN
     #statOverfirst:=1;
   // Z-parameters For Laplace PT1-System
   #statRe1 := - EXP(-#cycle/#tmLag1);
   #statRf1 := #gain*(1 + #statRe1);
   END_IF;

   // Differencial Equation of PT1-System
   #statOutput := #input*#statRf1 - #statOutput*#statRe1;

   // max limit of acutating variable
   IF #statOutput > #maxOut THEN
     #statOutput := #maxOut;
     #maxReached:= True;
   ELSE
     #maxReached := False;
   END_IF;

   // min limit of acutating variable
   IF #statOutput < #minOut THEN
     #statOutput := #minOut;
     #minReached := True;
   ELSE
     #minReached := False;
   END_IF;

   IF #reset THEN
     #statOutput := 0;
   END_IF;

   #output := #statOutput;
END_FUNCTION_BLOCK

FUNCTION_BLOCK "LSim_PT3"   // FB54, SCL
{ S7_Optimized_Access := 'TRUE' }
VERSION : 2.01
   VAR_INPUT
      input : Real;   // input variable
      tmLag1 : Real := 29.0;   // time lag 1 in s
      tmLag2 : Real := 17.5;   // time lag 2 in s
      tmLag3 : Real := 3.1;   // time lag 3 in s
      gain : Real := 1.0;   // proportional gain
      disturb : Real;   // disturbance variable (additional to "input")
      cycle : Real := 0.1;   // sample time [in sec]
      reset : Bool;   // complete restart (#output = #input)
   END_VAR
   VAR_OUTPUT
      error : Bool;   // error (#tmLag1 <= 0 or #tmLag2 <= 0 or #tmLag3 <= 0)
      status : Word;   // status (if #error = TRUE then status = 16#8001)
      output : Real;   // output signal (if #error = FALSE)
   END_VAR
   VAR
      statFback1 : Real;   // feedback path value 1
      statFback2 : Real;   // feedback path value 2
      statFback3 : Real;   // feedback path value 3
   END_VAR
   VAR_TEMP
      tempHvar : Real;   // help variable
      tempCycleR : Real;   // cycle to real
      tempTmLag1R : Real;   // time lag 1 to real
      tempTmLag2R : Real;   // time lag 2 to real
      tempTmLag3R : Real;   // time lag 3 to real
      tempOutvNew : Real;   // new output variable
   END_VAR
BEGIN
   //=============================================================================
   //SIEMENS AG
   //(c)Copyright 2017 All Rights Reserved
   //-----------------------------------------------------------------------------
   //Library:       Library for Controlled System Simulation
   //Tested with:   S7-1500 FW V2.0 / S7-1200 FW V4.2
   //Engineering:   STEP 7 V14 Upd2 (TIA Portal)
   //Restrictions:  Cyclic interrupt
   //Requirements:  memory card needed for S7-1500
   //Functionality: Simulation of an PT3-system
   //
   //                               gain
   //  F(p) = ------------------------------------------------------
   //         (tmLag1 * p + 1) * (tmLag2 * p + 1) * (tmLag3 * p + 1)
   //          
   //  Call the simulation in a cyclic interrupt with
   //  cyclic interrupt time at least = tmLag1/10!
   //-----------------------------------------------------------------------------
   //Change log table:
   //Version  Date       Expert in charge                Changes applied
   //02.00.00 03.02.2016 Siemens Industry Online Support Release (STEP 7 V13 SP1)
   //02.00.01 02.03.2017 Siemens Industry Online Support Release (STEP 7 V14)
   //=============================================================================
   // check parameter
   IF #tmLag1 <= 0 OR #tmLag2 <= 0 OR #tmLag3 <= 0 THEN
     #error := TRUE;
     #status := W#16#8001;     // Parameter Error
     #output := #input; //write output data
     #statFback1 := #input; //write static data
     #statFback2 := #input;
     #statFback3 := #input;
     RETURN;
   ELSE
     #error := FALSE;
     #status := W#16#0000;     // no error
   END_IF;

   IF #reset THEN //complete restart routine

     #output := #input;//write output data
     #statFback1 := #input;//write static data
     #statFback2 := #input;
     #statFback3 := #input;

   ELSE //cycle mode routine

     #tempCycleR  := #cycle*1000; //transform data type
     #tempTmLag1R := #tmLag1*1000;
     #tempTmLag2R := #tmLag2*1000;
     #tempTmLag3R := #tmLag3*1000;

     IF #tempCycleR * 0.5 > #tempTmLag1R THEN //limit TM_LAG1
       #tempTmLag1R := #tempCycleR * 0.5;
     END_IF;

     IF #tempCycleR * 0.5 > #tempTmLag2R THEN //limit TM_LAG2
       #tempTmLag2R := #tempCycleR * 0.5;
     END_IF;

     IF #tempCycleR * 0.5 > #tempTmLag3R THEN //limit TM_LAG2
       #tempTmLag3R := #tempCycleR * 0.5;
     END_IF;

     //1. first order lag algorithm
     #tempHvar     := #tempCycleR / (#tempTmLag1R * 2.0); 
     #tempHvar     := (#gain * (#input + #disturb) - #statFback1) * #tempHvar / (#tempHvar + 1.0);
     #tempOutvNew  := #tempHvar + #statFback1;
     #statFback1  := #tempHvar * 2.0 + #statFback1;

     //2. first order lag algorithm
     #tempHvar     := #tempCycleR / (#tempTmLag2R * 2.0); 
     #tempHvar     := ((#tempOutvNew - #statFback2) * #tempHvar) / (#tempHvar + 1.0);
     #tempOutvNew  := #tempHvar + #statFback2;
     #statFback2  := #tempHvar * 2.0 + #statFback2;

     //3. first order lag algorithm
     #tempHvar     := #tempCycleR / (#tempTmLag3R * 2.0); 
     #tempHvar     := ((#tempOutvNew - #statFback3) * #tempHvar) / (#tempHvar + 1.0);
     #tempOutvNew  := #tempHvar + #statFback3;
     #statFback3  := #tempHvar * 2.0 + #statFback3;

     #output := #tempOutvNew; //write output

   END_IF;
END_FUNCTION_BLOCK

FUNCTION_BLOCK "LSim_I"   // FB56, SCL
{ S7_Optimized_Access := 'TRUE' }
VERSION : 2.01
   VAR_INPUT
      calcParam : Bool;   // recalculate with new parameters
      input : Real;   // input signal
      tmLag1 : Real := 1.0;   // time constant T1 [sec]
      cycle : Real := 0.1;   // cyclic time [sec]
      maxOut : Real := 100.0;   // max. output limit
      minOut : Real;   // min. output limit
      reset : Bool;   // resets all relevant parameters to ‘0’ including the output
   END_VAR
   VAR_OUTPUT
      error : Bool;   // error (#tmLag1 <= 0)
      status : Word;   // status (if #tmLag1 <= 0 then status = 16#8001)
      maxReached : Bool;   // output has reached max. limit
      minReached : Bool;   // output has reached min. limit
      output : Real;   // output signal (if #error = FALSE)
   END_VAR
   VAR
      statRxn1 : Real;   // delayed input signal (n-1)
      statRyn1 : Real;   // delayed output signal (n-1)
      statRa1 : Real;
      statRb1 : Real;
      statOverfirst : Bool;
      statOutput : Real;   // output signal
   END_VAR
BEGIN
   //=============================================================================
   //SIEMENS AG
   //(c)Copyright 2017 All Rights Reserved
   //-----------------------------------------------------------------------------
   //Library:       Library for Controlled System Simulation
   //Tested with:   S7-1500 FW V2.0 / S7-1200 FW V4.2
   //Engineering:   STEP 7 V14 Upd2 (TIA Portal)
   //Restrictions:  Cyclic interrupt
   //Requirements:  memory card needed for S7-1500
   //Functionality: Simulation of a I-System
   //
   //             1
   //  F(p) = -----------
   //         (tmLag1*p)
   //          
   //  Call the simulation in a cyclic interrupt with
   //  cyclic interrupt time at least = tmLag1/10!
   //-----------------------------------------------------------------------------
   //Change log table:
   //Version  Date       Expert in charge                Changes applied
   //02.00.00 03.02.2016 Siemens Industry Online Support Release (STEP 7 V13 SP1)
   //02.00.01 02.03.2017 Siemens Industry Online Support Release (STEP 7 V14)
   //=============================================================================

   // check parameter
   IF #tmLag1 <= 0 THEN
     #error := True;
     #status := W#16#8001;     // Parameter Error
     #statRxn1 := 0.0;
     #statRyn1 := 0.0;
     #statOutput := 0;
     #output := 0;
     RETURN;
   ELSE
     #error := FALSE;
     #status := W#16#0000;     // no error
   END_IF;

   // calculates the z-parameter for the difference equatation
   IF #calcParam = True OR NOT #statOverfirst THEN
   #statOverfirst:=1;
     // Calculate z-parameters for IT1-System
   #statRb1 := #cycle/#tmLag1;
   #statRa1 := -1;

   END_IF;

   // reset Memory
   IF #reset = True THEN
     #statRxn1 := 0.0;
     #statRyn1 := 0.0;
     #statOutput:=0;
   END_IF;

   // save delayed output-signals
   #statRyn1:= #statOutput;

   // difference equatation for the I-system
   #statOutput := #statRxn1* #statRb1 - #statRyn1*#statRa1;

   // save delayed input-signals
   #statRxn1 := #input;

   // max limit of acutating variable
   IF #statOutput > #maxOut THEN
     #statOutput := #maxOut;
     #maxReached:= True;
   ELSE
     #maxReached := False;
   END_IF;

   // min limit of acutating variable
   IF #statOutput < #minOut THEN
     #statOutput := #minOut;
     #minReached := True;
   ELSE
     #minReached := False;
   END_IF;

   #output := #statOutput;
END_FUNCTION_BLOCK

FUNCTION "FC_2_GetStringSizeOfNumber" : Void   // FC1, SCL
{ S7_Optimized_Access := 'TRUE' }
VERSION : 0.1
   VAR_INPUT
      number : UDInt;
   END_VAR
   VAR_OUTPUT
      stringSize : Int;
   END_VAR
   VAR_TEMP
      size : USInt;
   END_VAR
BEGIN
   IF #number < 10 THEN
       #size := 1;
   ELSIF #number >= 10 AND #number < 100 THEN
       #size := 2;
   ELSIF #number >= 100 AND #number < 1000 THEN
       #size := 3;
   ELSIF #number >= 1000 AND #number < 10000 THEN
       #size := 4;
   ELSIF #number >= 10000 AND #number < 100000 THEN
       #size := 5;
   ELSIF #number >= 100000 AND #number < 1000000 THEN
       #size := 6;
   ELSIF #number >= 1000000 AND #number < 10000000 THEN
       #size := 7;
   ELSIF #number >= 10000000 AND #number < 100000000 THEN
       #size := 8;
   ELSIF #number >= 100000000 AND #number < 1000000000 THEN
       #size := 9;
   ELSIF #number >= 1000000000 AND #number < 10000000000 THEN
       #size := 10;
   ELSE    // max UDINT = 4.294.967.295
       #size := 11;
   END_IF;
END_FUNCTION

FUNCTION "FC_1_Random_Number" : Void   // FC3, SCL
{ S7_Optimized_Access := 'TRUE' }
VERSION : 0.1
   VAR_INPUT
      Min : UDInt;
      Max : UDInt;
   END_VAR
   VAR_OUTPUT
      RandomNumber : UDInt;
   END_VAR
   VAR_TEMP
      range : UDInt;
      tmp : UDInt;
   END_VAR
BEGIN
   // generate random number
   #tmp := DINT_TO_UDINT(TIME_TO_DINT(TIME_TCK()));

   IF #tmp < 0 THEN
       #tmp := #tmp * - 1;
   END_IF;

   "Manipulator" := "Manipulator" + 1;

   IF "Manipulator" = 10 THEN
       "Manipulator" := 1;
   END_IF;

   #tmp := #tmp / "Manipulator";

   #range := #Max - #Min;

   #tmp := #tmp MOD (#range + 1);
   #RandomNumber := #tmp + #Min;
END_FUNCTION

ORGANIZATION_BLOCK "Main"   // OB1, LAD, ProgramCycle
TITLE = "Main Program Sweep (Cycle)"
{ S7_Optimized_Access := 'TRUE' }
VERSION : 0.1
   VAR_INPUT
      Initial_Call : Bool;   // Initial call of this OB
      Remanence : Bool;   // =True, if remanent data are available
   END_VAR
BEGIN
END_ORGANIZATION_BLOCK

ORGANIZATION_BLOCK "Cyclic interrupt"   // OB30, FBD, CyclicInterrupt
{ S7_Optimized_Access := 'TRUE' }
VERSION : 0.1
   VAR_INPUT
      Initial_Call : Bool;   // Initial call of this OB
      Event_Count : Int;   // Events discarded
   END_VAR
   VAR_TEMP
      tempStopCip : Bool;   // stop CIP S7 graph sequence
      tempStartCip : Bool;   // start CIP S7 graph sequence
   END_VAR
BEGIN

REGION Network 1: call filling sequence
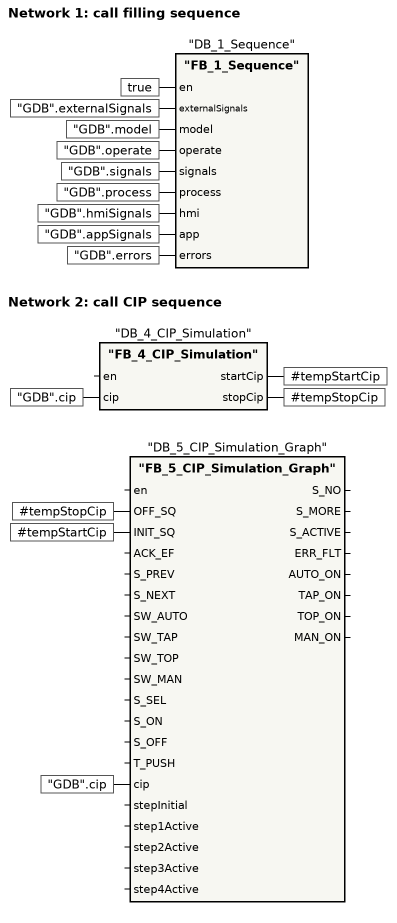
   IF true THEN
       "DB_1_Sequence"(externalSignals := "GDB".externalSignals,   // "FB_1_Sequence"
                       model := "GDB".model,
                       operate := "GDB".operate,
                       signals := "GDB".signals,
                       process := "GDB".process,
                       hmi := "GDB".hmiSignals,
                       app := "GDB".appSignals,
                       errors := "GDB".errors);
   END_IF;
END_REGION

REGION Network 2: call CIP sequence
   "DB_4_CIP_Simulation"(cip := "GDB".cip, startCip => #tempStartCip, stopCip => #tempStopCip);   // "FB_4_CIP_Simulation"
   "DB_5_CIP_Simulation_Graph"(OFF_SQ := #tempStopCip, INIT_SQ := #tempStartCip, cip := "GDB".cip);   // "FB_5_CIP_Simulation_Graph"
END_REGION
END_ORGANIZATION_BLOCK

ORGANIZATION_BLOCK "ProDiagOB"   // OB250, ProDiag_OB, ProgramCycle
TITLE = "Main Program Sweep (Cycle)"
{ S7_Optimized_Access := 'TRUE' }
VERSION : 0.1
   VAR_INPUT
      Initial_Call : Bool;   // Initial call of this OB
      Remanence : Bool;   // =True, if remanent data are available
   END_VAR
BEGIN

REGION Network 1
   CALL "FB_Prodiag", "Block_1_DB";
END_REGION
END_ORGANIZATION_BLOCK

// folder: LGF/06 Converter operations

FUNCTION "LGF_DTLToString_ISO" : String   // FC10083, SCL
TITLE = LGF_DTLtoString_ISO
{ S7_Optimized_Access := 'TRUE' }
AUTHOR : Siemens_Digital_Industry
FAMILY : LGF
NAME : LGF_DTLtoString_ISO
// This function converts a date of data type DTL into a character string of data type STRING in international format (YYYY MM DD…). / Diese Funktion konvertiert ein Datum vom Datentyp DTL in eine Zeichenkette vom Datentyp STRING im internationalen Format (YYYY MM DD ...).
   VAR_INPUT
      "date" : DTL;   // Date to convert as DTL tag / Datum zum Konvertieren im Format DTL
      separator : Char;   // Separator between the components of the output date. / Trennzeichen zwischen den Komponenten des ausgegebenen Datums.
   END_VAR
   VAR_TEMP
      tempString : String;   // Temp string to setup the date string
      tempIndex : DInt;   // Temp iterator for replacing withspaces with '0' in nanosecondstring
   END_VAR
   // Ret_Val : Output string in accordance with the ISO 8601 format. Example: `2019-01-22 14:06:51.524621000`. / Ausgegebenen Zeichenkette entsprechend dem Format ISO 8601. Beispiel: `2019-01-22 14:06:51.524621000`.
   VAR CONSTANT
      CONVERT_SIZE_YEAR : USInt := 4;   // Number of character positions for Year
      CONVERT_SIZE_MONTH_DAY_HOUR_MINUTE_SECOND : USInt := 2;   // Number of character positions for Month, Day, Minute and Second
      CONVERT_SIZE_NANOSECOND : USInt := 9;   // Number of character positions for Nanoseconds
      CONVERT_PRECISION : USInt := 0;   // Number of decimal places to convert
      CONVERT_FORMAT_TO_STRING : Word := 16#0000;   // Output format of the characters
      CONVERT_START_POSITION_YEAR : UInt := 1;   // Character starting in string at which position the result is written.
      CONVERT_START_POSITION_MONTH : UInt := 6;   // Character starting in string at which position the result is written.
      CONVERT_START_POSITION_DAY : UInt := 9;   // Character starting in string at which position the result is written.
      CONVERT_START_POSITION_HOUR : UInt := 12;   // Character starting in string at which position the result is written.
      CONVERT_START_POSITION_MINUTE : UInt := 15;   // Character starting in string at which position the result is written.
      CONVERT_START_POSITION_SECOND : UInt := 18;   // Character starting in string at which position the result is written.
      CONVERT_START_POSITION_NANOSECOND : UInt := 21;   // Character starting in string at which position the result is written.
      SEPARATOR_POSITION_YEAR_MONTH : UInt := 5;   // Character starting in string at which position the result is written.
      SEPARATOR_POSITION_MONTH_DAY : UInt := 8;   // Character starting in string at which position the result is written.
      SEPARATOR_POSITION_HOUR_MINUTE : UInt := 14;   // Character starting in string at which position the result is written.
      SEPARATOR_POSITION_MINUTE_SECOND : UInt := 17;   // Character starting in string at which position the result is written.
      SEPARATOR_POSITION_SECOND_NANOSECOND : UInt := 20;   // Character starting in string at which position the result is written.
      SEPARATOR_NANOSECOND : Char := '.';   // Seperator for Nanosecond
      SEPARATOR_TIME : Char := ':';   // Seperator for Time
      SEPARATOR_DATE : Char := '-';   // Default separator for Date
      REPLACE_NANOSECOND_COUNT : DInt := 8;   // Number of Nonosecond characters to be checked for replacing withspaces wit '0'
   END_VAR
BEGIN
   REGION BLOCK INFO HEADER
     //===============================================================================
     // SIEMENS AG / (c)Copyright 2019
     //-------------------------------------------------------------------------------
     // Title:            LGF_DTLtoString_ISO
     // Comment/Function: This function converts a date of data type DTL into a character string of data type STRING in international format (YYYY MM DD…).
     // Library/Family:   LGF (Library General Functions)
     // Author:           Siemens Digital Industry Support
     // Tested with:      S7-PLCSIM Advanced V2.0 SP1
     // Engineering:      TIA Portal V15.1
     // Restrictions:     ENO mechanism is not used, no error handling
     // Requirements:     PLC (S7-1200 / S7-1500)
     //-------------------------------------------------------------------------------
     // Change log table:
     // Version  | Date       | Expert in charge       | Changes applied
     //----------|------------|------------------------|------------------------------
     // 01.00.00 | 15.06.2016 | Siemens Industry Online Support
     //                         First released version
     // 01.00.01 | 02.01.2017 | Siemens Industry Online Support
     //                         Upgrade: TIA Portal V14 Update 1
     // 01.00.02 | 17.08.2018 | Siemens Industry Online Support
     //                         Upgrade: TIA V15 Update 2
     // 01.00.03 | 23.11.2018 | Siemens Industry Online Support
     //                         Upgrade: TIA V15.1
     // 01.00.04 | 17.07.2019 | Simatic Systems Support
     //                         Bugfix - nanosecond precision and '0' filling
     // 01.00.05 | 18.07.2019 | Simatic Systems Support
     //                         Renamed from "LGF_DTLtoString" to "LGF_DTLtoString_ISO"
     //                         Split into two blocks, removed "format" input
     // 03.00.00 | 23.04.2020 | Simatic Systems Support | Set version to V3.0.0
     //                         Harmonize the version of the whole library
     // 03.00.01 | 23.02.2021 | Simatic Systems Support
     //                         Insert documentation
     //=============================================================================
   END_REGION Block info header

   REGION DESCRIPTION
     (/*The block reads a date of data type DTL and converts the individual components of the date (year, month, day, hour…) into a character string and outputs it in international format. The separator between the components of the date is variable.

   ##### International format (ISO 8601):

   {.imagePageWidth}
   ![LGF_DTLtoString_ISO - Structure of the character string in accordance with ISO 8601](LGF_DTLtoString_ISO.png "LGF_DTLtoString_ISO - Structure of the character string in accordance with ISO 8601")

   ##### Separator:

   At the input parameter `separatorDate`, you specify the separator between the components of the calendar date.

   ##### Example:

   * separatorDate = `/` - outString = `2016/03/16…`
   * separatorDate = `-` - outString = `2016-03-16…`
   Der Baustein liest ein Datum vom Datentyp DTL ein und konvertiert die einzelnen Komponenten des Datums (Jahr, Monat, Tag, Stunde...) in eine Zeichenkette und gibt diese im internationalen Format aus. Das Trennzeichen zwischen den Komponenten des Datums ist variabel.

   ##### Internationales Format (ISO 8601):

